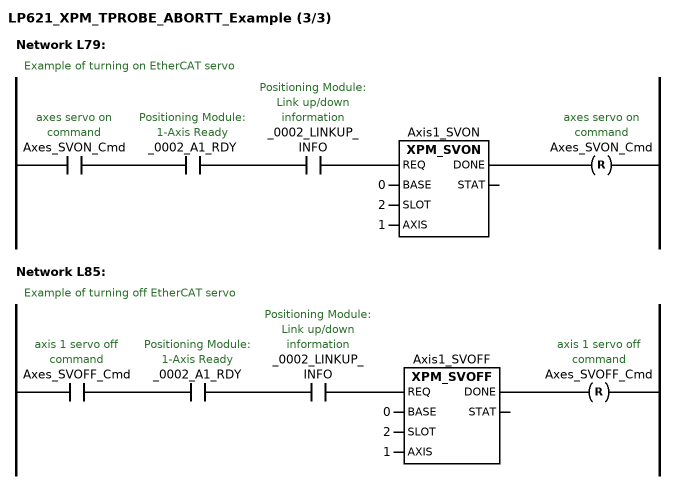
(* [picture p24: LP621_XPM_TPROBE_ABORTT_Example rungs L79-L85] *)
(* Example of turning on EtherCAT servo *)
(* Rung L79 *)
Axis1_SVON(REQ := Axes_SVON_Cmd AND _0002_A1_RDY AND _0002_LINKUP_INFO, BASE := 0, SLOT := 2, AXIS := 1);
IF Axis1_SVON.DONE THEN Axes_SVON_Cmd := FALSE; END_IF;
(* Example of turning off EtherCAT servo *)
(* Rung L85 *)
Axis1_SVOFF(REQ := Axes_SVOFF_Cmd AND _0002_A1_RDY AND _0002_LINKUP_INFO, BASE := 0, SLOT := 2, AXIS := 1);
IF Axis1_SVOFF.DONE THEN Axes_SVOFF_Cmd := FALSE; END_IF;
END_PROGRAM

PROGRAM LP622_Read_Data_Example (* task: Scan Program *)
(* example program for XPM_CRD and XPM_SRD function blocks. *)
VAR
    Axes_SVOFF_Cmd : BOOL; (* axis 1 servo off command *)
    Axes_SVON_Cmd : BOOL; (* axes servo on command *)
    Axis1_Commanded_Position : DINT; (* commanded position of axis 1 *)
    Axis1_Commanded_Speed : DINT; (* commanded speed of axis 1 *)
    Axis1_CommonError_Number : UINT; (* common error number for axis 1 *)
    Axis1_CRD : XPM_CRD; (* axis 1 drive information fb *)
    Axis1_Current_Position : DINT; (* current position of axis 1 *)
    Axis1_Current_Speed : DINT; (* current speed of axis 1 *)
    Axis1_Current_Step : UINT; (* current position table step of axis 1 *)
    Axis1_Current_Torque : INT; (* current torque of axis 1 *)
    Axis1_Error_Number : UINT; (* error number for axis 1 *)
    Axis1_MCode : UINT; (* axis1 mcode *)
    Axis1_Read_Data : BOOL; (* command to read axis data *)
    Axis1_SRD : XPM_SRD; (* axis 1 state function block *)
    Axis1_ST1 : ARRAY[0..7] OF BOOL; (* axis 1 state 1 information *)
    Axis1_ST2 : ARRAY[0..7] OF BOOL; (* axis 1 state 2 information *)
    Axis1_ST3 : ARRAY[0..7] OF BOOL; (* axis 1 state 3 information *)
    Axis1_ST4 : ARRAY[0..7] OF BOOL; (* axis 1 state 4 information *)
    Axis1_ST5 : ARRAY[0..7] OF BOOL; (* axis 1 state 5 information *)
    Axis1_ST6 : ARRAY[0..7] OF BOOL; (* axis 1 state 6 information *)
    Axis1_ST7 : ARRAY[0..7] OF BOOL; (* axis 1 state 7 information *)
    Axis1_SVOFF : XPM_SVOFF; (* function block for axis 1 servo off *)
    Axis1_SVON : XPM_SVON; (* SVON fb for axis 1 *)
    Connect_Servos : BOOL; (* command to connect to ECAT servos *)
    DCON_FB : XPM_DCON; (* EtherCAT disconnect FB *)
    Disconnect_Servos : BOOL; (* Disconnect from ECAT servos *)
    ECON_FB : XPM_ECON; (* EtherCAT connect FB *)
END_VAR
VAR_EXTERNAL
    _0002_A1_RDY : BOOL; (* AT %UX0.2.0 *) (* Positioning Module: 1-Axis Ready *)
    _0002_LINKUP_INFO : BOOL; (* AT %UX0.2.14 *) (* Positioning Module: Link up/down information *)
END_VAR

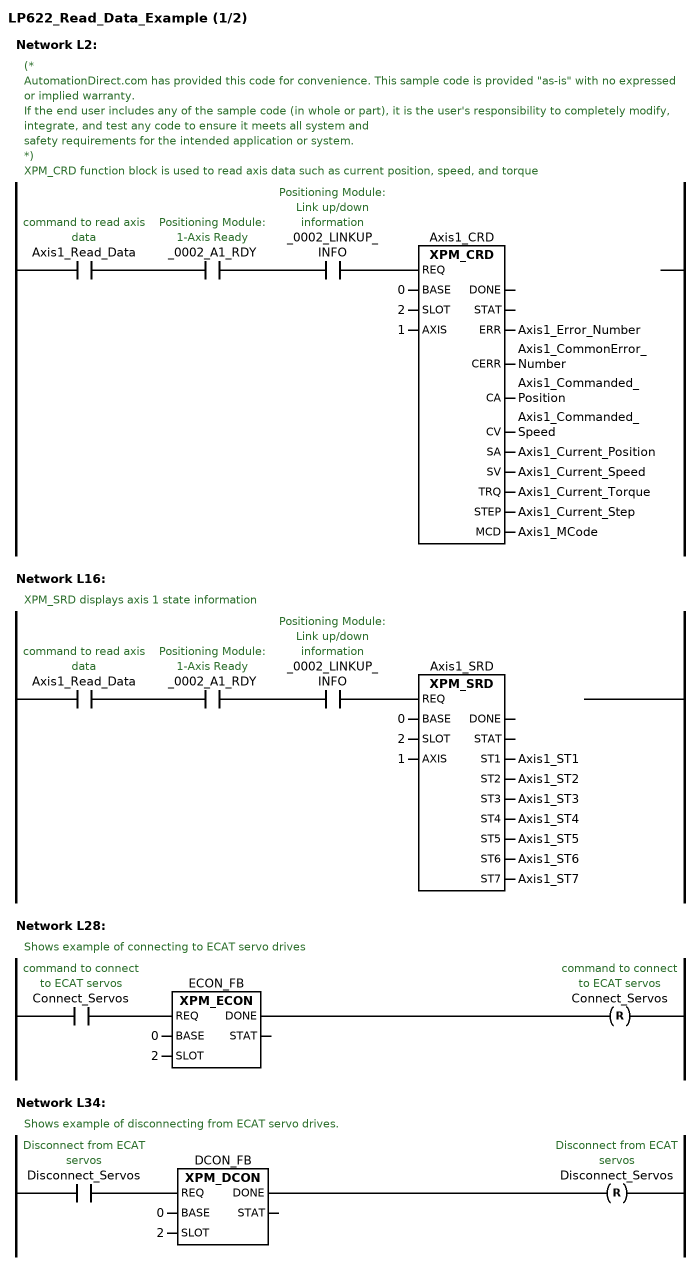
(* ( * / AutomationDirect.com has provided this code for convenience. This sample code is provided "as-is" with no expressed or implied warranty. / If the end user includes any of the sample code (in whole or part), it is the user's responsibility to completely modify, integrate, and test any code to ensure it meets all system and / safety requirements for the intended application or system. / * ) *)
(* XPM_CRD function block is used to read axis data such as current position, speed, and torque *)
(* Rung L2 *)
Axis1_CRD(REQ := Axis1_Read_Data AND _0002_A1_RDY AND _0002_LINKUP_INFO, BASE := 0, SLOT := 2, AXIS := 1, ERR => Axis1_Error_Number, CERR => Axis1_CommonError_Number, CA => Axis1_Commanded_Position, CV => Axis1_Commanded_Speed, SA => Axis1_Current_Position, SV => Axis1_Current_Speed, TRQ => Axis1_Current_Torque, STEP => Axis1_Current_Step, MCD => Axis1_MCode);
(* XPM_SRD displays axis 1 state information *)
(* Rung L16 *)
Axis1_SRD(REQ := Axis1_Read_Data AND _0002_A1_RDY AND _0002_LINKUP_INFO, BASE := 0, SLOT := 2, AXIS := 1, ST1 => Axis1_ST1, ST2 => Axis1_ST2, ST3 => Axis1_ST3, ST4 => Axis1_ST4, ST5 => Axis1_ST5, ST6 => Axis1_ST6, ST7 => Axis1_ST7);
(* Shows example of connecting to ECAT servo drives *)
(* Rung L28 *)
ECON_FB(REQ := Connect_Servos, BASE := 0, SLOT := 2);
IF ECON_FB.DONE THEN Connect_Servos := FALSE; END_IF;
(* Shows example of disconnecting from ECAT servo drives. *)
(* Rung L34 *)
DCON_FB(REQ := Disconnect_Servos, BASE := 0, SLOT := 2);
IF DCON_FB.DONE THEN Disconnect_Servos := FALSE; END_IF;

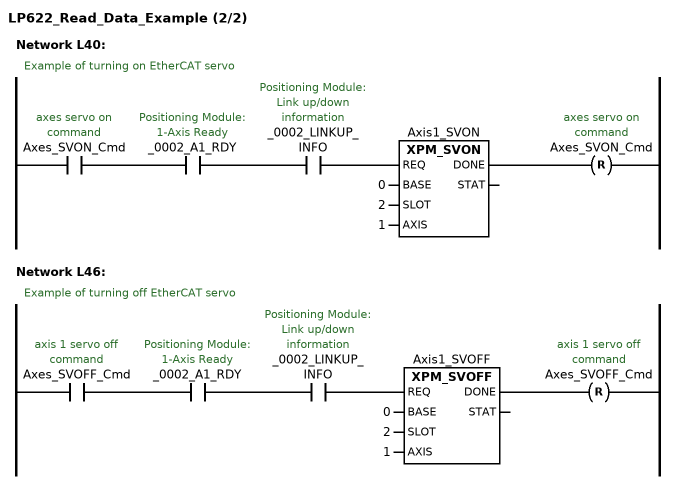
(* Example of turning on EtherCAT servo *)
(* Rung L40 *)
Axis1_SVON(REQ := Axes_SVON_Cmd AND _0002_A1_RDY AND _0002_LINKUP_INFO, BASE := 0, SLOT := 2, AXIS := 1);
IF Axis1_SVON.DONE THEN Axes_SVON_Cmd := FALSE; END_IF;
(* Example of turning off EtherCAT servo *)
(* Rung L46 *)
Axis1_SVOFF(REQ := Axes_SVOFF_Cmd AND _0002_A1_RDY AND _0002_LINKUP_INFO, BASE := 0, SLOT := 2, AXIS := 1);
IF Axis1_SVOFF.DONE THEN Axes_SVOFF_Cmd := FALSE; END_IF;
END_PROGRAM

PROGRAM LP624_XPM_JOG_Example (* task: Scan Program *)
(* example program for XPM_JOG and XPM_RTP function block. *)
VAR
    Axes_SVOFF_Cmd : BOOL; (* axis 1 servo off command *)
    Axes_SVON_Cmd : BOOL; (* axes servo on command *)
    Axis1_Home : XPM_FLT; (* direct home of axis 1 *)
    Axis1_Jog_FWD : XPM_JOG; (* fb to jog axis 1 fwd *)
    Axis1_Jog_FWD_CMD : BOOL; (* command to jog axis 1 forward *)
    Axis1_Jog_REV : XPM_JOG; (* axis 1 jog reverse fb *)
    Axis1_Jog_REV_CMD : BOOL; (* command to jog axis 1 in reverse *)
    Axis1_RTP : XPM_RTP; (* axis 1 return to position fb *)
    Axis1_RTP_CMD : BOOL; (* return axis 1 to position before manual move *)
    Axis1_SVOFF : XPM_SVOFF; (* function block for axis 1 servo off *)
    Axis1_SVON : XPM_SVON; (* SVON fb for axis 1 *)
    Axis2_Jog_FWD : XPM_JOG; (* fb to jog axis 1 fwd *)
    Connect_Servos : BOOL; (* command to connect to ECAT servos *)
    DCON_FB : XPM_DCON; (* EtherCAT disconnect FB *)
    Disconnect_Servos : BOOL; (* Disconnect from ECAT servos *)
    ECON_FB : XPM_ECON; (* EtherCAT connect FB *)
    Home_Axes : BOOL; (* home the axes *)
END_VAR
VAR_EXTERNAL
    _0002_A1_RDY : BOOL; (* AT %UX0.2.0 *) (* Positioning Module: 1-Axis Ready *)
    _0002_A4_RDY : BOOL; (* AT %UX0.2.3 *) (* Positioning Module: 4-Axis Ready *)
    _0002_LINKUP_INFO : BOOL; (* AT %UX0.2.14 *) (* Positioning Module: Link up/down information *)
END_VAR

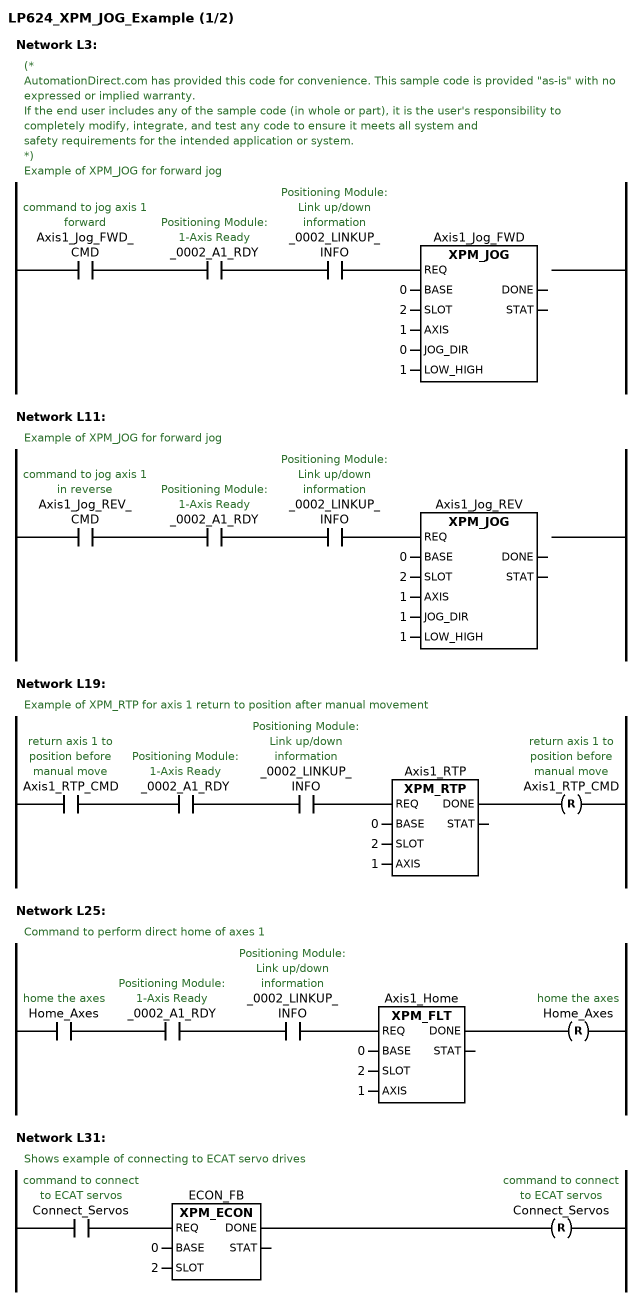
(* ( * / AutomationDirect.com has provided this code for convenience. This sample code is provided "as-is" with no expressed or implied warranty. / If the end user includes any of the sample code (in whole or part), it is the user's responsibility to completely modify, integrate, and test any code to ensure it meets all system and / safety requirements for the intended application or system. / * ) *)
(* Example of XPM_JOG for forward jog *)
(* Rung L3 *)
Axis1_Jog_FWD(REQ := Axis1_Jog_FWD_CMD AND _0002_A1_RDY AND _0002_LINKUP_INFO, BASE := 0, SLOT := 2, AXIS := 1, JOG_DIR := 0, LOW_HIGH := 1);
(* Example of XPM_JOG for forward jog *)
(* Rung L11 *)
Axis1_Jog_REV(REQ := Axis1_Jog_REV_CMD AND _0002_A1_RDY AND _0002_LINKUP_INFO, BASE := 0, SLOT := 2, AXIS := 1, JOG_DIR := 1, LOW_HIGH := 1);
(* Example of XPM_RTP for axis 1 return to position after manual movement *)
(* Rung L19 *)
Axis1_RTP(REQ := Axis1_RTP_CMD AND _0002_A1_RDY AND _0002_LINKUP_INFO, BASE := 0, SLOT := 2, AXIS := 1);
IF Axis1_RTP.DONE THEN Axis1_RTP_CMD := FALSE; END_IF;
(* Command to perform direct home of axes 1 *)
(* Rung L25 *)
Axis1_Home(REQ := Home_Axes AND _0002_A1_RDY AND _0002_LINKUP_INFO, BASE := 0, SLOT := 2, AXIS := 1);
IF Axis1_Home.DONE THEN Home_Axes := FALSE; END_IF;
(* Shows example of connecting to ECAT servo drives *)
(* Rung L31 *)
ECON_FB(REQ := Connect_Servos, BASE := 0, SLOT := 2);
IF ECON_FB.DONE THEN Connect_Servos := FALSE; END_IF;

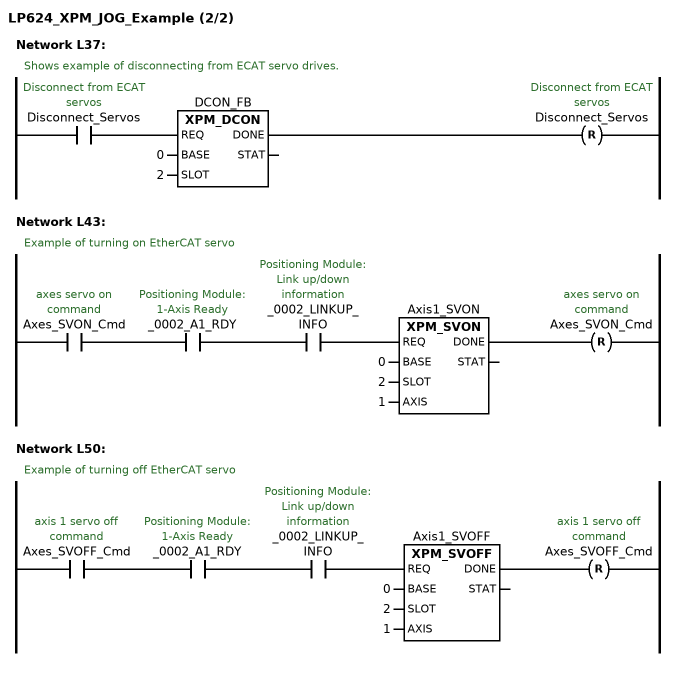
(* Shows example of disconnecting from ECAT servo drives. *)
(* Rung L37 *)
DCON_FB(REQ := Disconnect_Servos, BASE := 0, SLOT := 2);
IF DCON_FB.DONE THEN Disconnect_Servos := FALSE; END_IF;
(* Example of turning on EtherCAT servo *)
(* Rung L43 *)
Axis1_SVON(REQ := Axes_SVON_Cmd AND _0002_A1_RDY AND _0002_LINKUP_INFO, BASE := 0, SLOT := 2, AXIS := 1);
IF Axis1_SVON.DONE THEN Axes_SVON_Cmd := FALSE; END_IF;
(* Example of turning off EtherCAT servo *)
(* Rung L50 *)
Axis1_SVOFF(REQ := Axes_SVOFF_Cmd AND _0002_A1_RDY AND _0002_LINKUP_INFO, BASE := 0, SLOT := 2, AXIS := 1);
IF Axis1_SVOFF.DONE THEN Axes_SVOFF_Cmd := FALSE; END_IF;
END_PROGRAM

PROGRAM LP625_XPM_INC_Example (* task: Scan Program *)
(* example program for XPM_INC and XPM_RTP function block. *)
VAR
    Axes_SVOFF_Cmd : BOOL; (* axis 1 servo off command *)
    Axes_SVON_Cmd : BOOL; (* axes servo on command *)
    Axis1_Home : XPM_FLT; (* direct home of axis 1 *)
    Axis1_Inch_CMD : BOOL; (* command to jog axis 1 forward *)
    Axis1_Inch_FB : XPM_INC; (* inching fb for axis 1 *)
    Axis1_Inch_Value : DINT; (* inching value for axis 1 *)
    Axis1_RTP : XPM_RTP; (* axis 1 return to position fb *)
    Axis1_RTP_CMD : BOOL; (* return axis 1 to position before manual move *)
    Axis1_SVOFF : XPM_SVOFF; (* function block for axis 1 servo off *)
    Axis1_SVON : XPM_SVON; (* SVON fb for axis 1 *)
    Connect_Servos : BOOL; (* command to connect to ECAT servos *)
    DCON_FB : XPM_DCON; (* EtherCAT disconnect FB *)
    Disconnect_Servos : BOOL; (* Disconnect from ECAT servos *)
    ECON_FB : XPM_ECON; (* EtherCAT connect FB *)
    Home_Axes : BOOL; (* home the axes *)
END_VAR
VAR_EXTERNAL
    _0002_A1_RDY : BOOL; (* AT %UX0.2.0 *) (* Positioning Module: 1-Axis Ready *)
    _0002_LINKUP_INFO : BOOL; (* AT %UX0.2.14 *) (* Positioning Module: Link up/down information *)
END_VAR

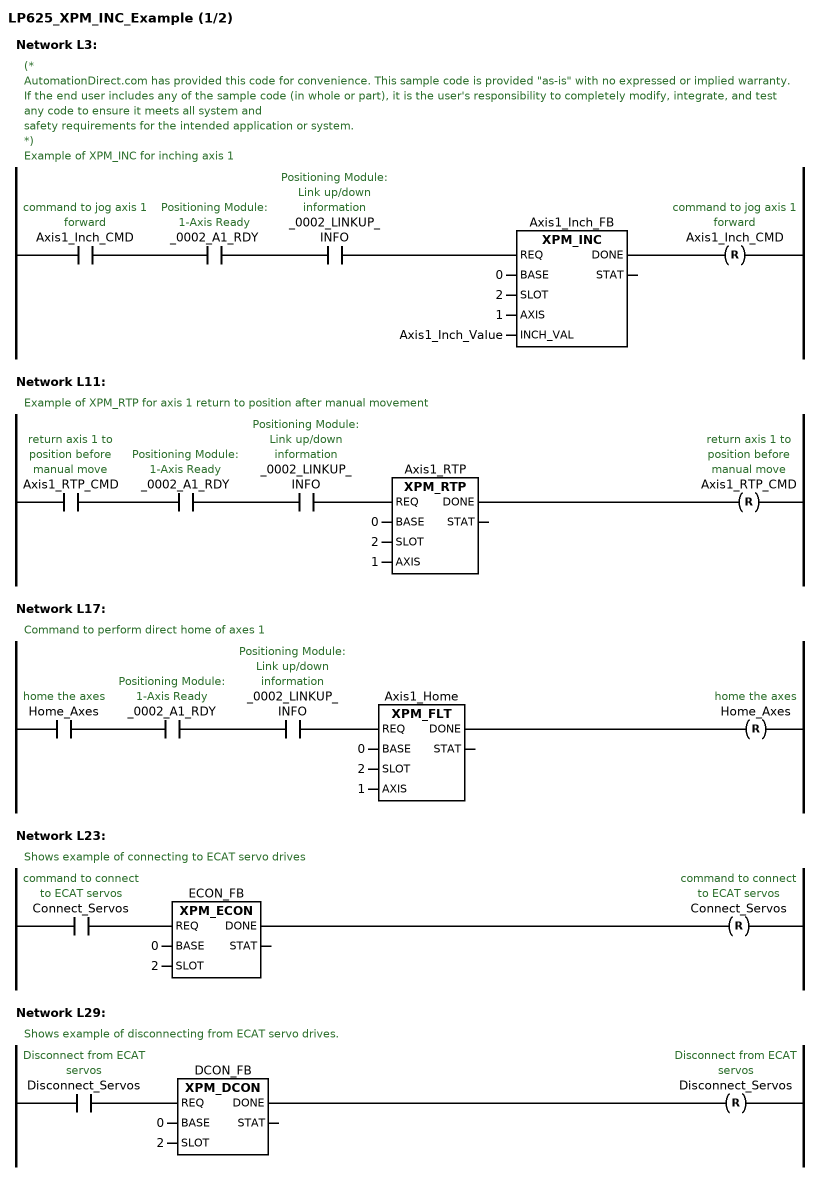
(* ( * / AutomationDirect.com has provided this code for convenience. This sample code is provided "as-is" with no expressed or implied warranty. / If the end user includes any of the sample code (in whole or part), it is the user's responsibility to completely modify, integrate, and test any code to ensure it meets all system and / safety requirements for the intended application or system. / * ) *)
(* Example of XPM_INC for inching axis 1 *)
(* Rung L3 *)
Axis1_Inch_FB(REQ := Axis1_Inch_CMD AND _0002_A1_RDY AND _0002_LINKUP_INFO, BASE := 0, SLOT := 2, AXIS := 1, INCH_VAL := Axis1_Inch_Value);
IF Axis1_Inch_FB.DONE THEN Axis1_Inch_CMD := FALSE; END_IF;
(* Example of XPM_RTP for axis 1 return to position after manual movement *)
(* Rung L11 *)
Axis1_RTP(REQ := Axis1_RTP_CMD AND _0002_A1_RDY AND _0002_LINKUP_INFO, BASE := 0, SLOT := 2, AXIS := 1);
IF Axis1_RTP.DONE THEN Axis1_RTP_CMD := FALSE; END_IF;
(* Command to perform direct home of axes 1 *)
(* Rung L17 *)
Axis1_Home(REQ := Home_Axes AND _0002_A1_RDY AND _0002_LINKUP_INFO, BASE := 0, SLOT := 2, AXIS := 1);
IF Axis1_Home.DONE THEN Home_Axes := FALSE; END_IF;
(* Shows example of connecting to ECAT servo drives *)
(* Rung L23 *)
ECON_FB(REQ := Connect_Servos, BASE := 0, SLOT := 2);
IF ECON_FB.DONE THEN Connect_Servos := FALSE; END_IF;
(* Shows example of disconnecting from ECAT servo drives. *)
(* Rung L29 *)
DCON_FB(REQ := Disconnect_Servos, BASE := 0, SLOT := 2);
IF DCON_FB.DONE THEN Disconnect_Servos := FALSE; END_IF;

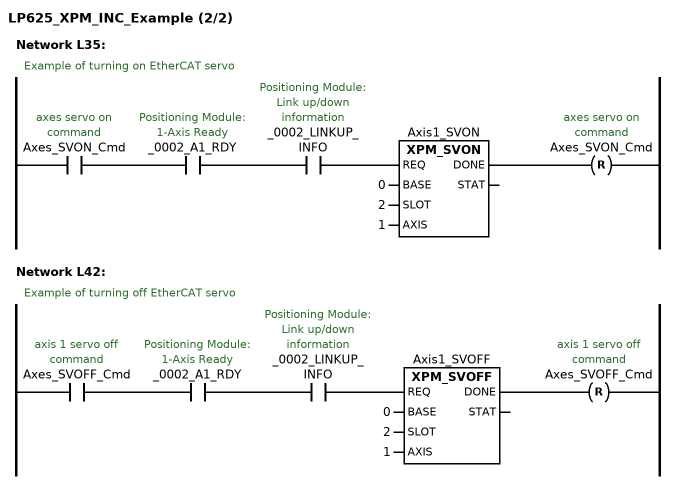
(* Example of turning on EtherCAT servo *)
(* Rung L35 *)
Axis1_SVON(REQ := Axes_SVON_Cmd AND _0002_A1_RDY AND _0002_LINKUP_INFO, BASE := 0, SLOT := 2, AXIS := 1);
IF Axis1_SVON.DONE THEN Axes_SVON_Cmd := FALSE; END_IF;
(* Example of turning off EtherCAT servo *)
(* Rung L42 *)
Axis1_SVOFF(REQ := Axes_SVOFF_Cmd AND _0002_A1_RDY AND _0002_LINKUP_INFO, BASE := 0, SLOT := 2, AXIS := 1);
IF Axis1_SVOFF.DONE THEN Axes_SVOFF_Cmd := FALSE; END_IF;
END_PROGRAM

PROGRAM LP626_Homing_Example (* task: Scan Program *)
(* example program for XPM_ORG and XPM_FLT  function block. *)
VAR
    Axes_SVOFF_Cmd : BOOL; (* axis 1 servo off command *)
    Axes_SVON_Cmd : BOOL; (* axes servo on command *)
    Axis1_FLT_CMD : BOOL; (* home axis 1 with XPM_FLT *)
    Axis1_ORG_CMD : BOOL; (* home axis 1 with XPM_ORG *)
    Axis1_SVOFF : XPM_SVOFF; (* function block for axis 1 servo off *)
    Axis1_SVON : XPM_SVON; (* SVON fb for axis 1 *)
    Axis1_XPM_FLT : XPM_FLT; (* direct home of axis 1 *)
    Axis1_XPM_ORG : XPM_ORG; (* axis 1 xpm_org fb *)
    Connect_Servos : BOOL; (* command to connect to ECAT servos *)
    DCON_FB : XPM_DCON; (* EtherCAT disconnect FB *)
    Disconnect_Servos : BOOL; (* Disconnect from ECAT servos *)
    ECON_FB : XPM_ECON; (* EtherCAT connect FB *)
END_VAR
VAR_EXTERNAL
    _0002_A1_RDY : BOOL; (* AT %UX0.2.0 *) (* Positioning Module: 1-Axis Ready *)
    _0002_LINKUP_INFO : BOOL; (* AT %UX0.2.14 *) (* Positioning Module: Link up/down information *)
END_VAR

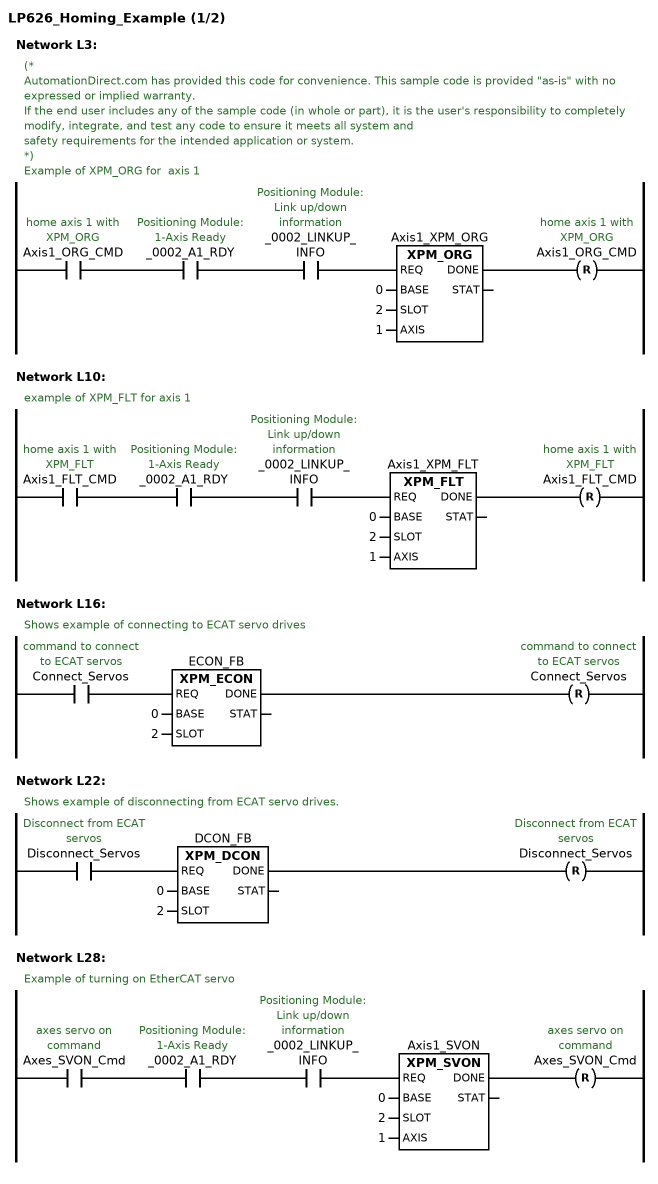
(* ( * / AutomationDirect.com has provided this code for convenience. This sample code is provided "as-is" with no expressed or implied warranty. / If the end user includes any of the sample code (in whole or part), it is the user's responsibility to completely modify, integrate, and test any code to ensure it meets all system and / safety requirements for the intended application or system. / * ) *)
(* Example of XPM_ORG for  axis 1 *)
(* Rung L3 *)
Axis1_XPM_ORG(REQ := Axis1_ORG_CMD AND _0002_A1_RDY AND _0002_LINKUP_INFO, BASE := 0, SLOT := 2, AXIS := 1);
IF Axis1_XPM_ORG.DONE THEN Axis1_ORG_CMD := FALSE; END_IF;
(* example of XPM_FLT for axis 1 *)
(* Rung L10 *)
Axis1_XPM_FLT(REQ := Axis1_FLT_CMD AND _0002_A1_RDY AND _0002_LINKUP_INFO, BASE := 0, SLOT := 2, AXIS := 1);
IF Axis1_XPM_FLT.DONE THEN Axis1_FLT_CMD := FALSE; END_IF;
(* Shows example of connecting to ECAT servo drives *)
(* Rung L16 *)
ECON_FB(REQ := Connect_Servos, BASE := 0, SLOT := 2);
IF ECON_FB.DONE THEN Connect_Servos := FALSE; END_IF;
(* Shows example of disconnecting from ECAT servo drives. *)
(* Rung L22 *)
DCON_FB(REQ := Disconnect_Servos, BASE := 0, SLOT := 2);
IF DCON_FB.DONE THEN Disconnect_Servos := FALSE; END_IF;
(* Example of turning on EtherCAT servo *)
(* Rung L28 *)
Axis1_SVON(REQ := Axes_SVON_Cmd AND _0002_A1_RDY AND _0002_LINKUP_INFO, BASE := 0, SLOT := 2, AXIS := 1);
IF Axis1_SVON.DONE THEN Axes_SVON_Cmd := FALSE; END_IF;

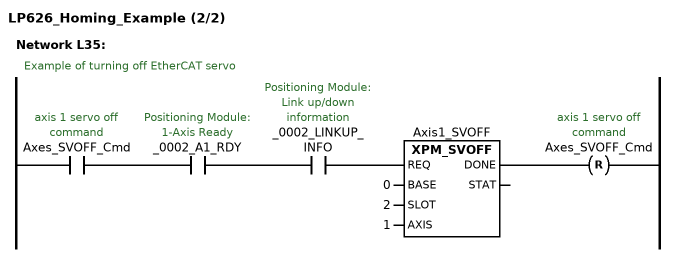
(* Example of turning off EtherCAT servo *)
(* Rung L35 *)
Axis1_SVOFF(REQ := Axes_SVOFF_Cmd AND _0002_A1_RDY AND _0002_LINKUP_INFO, BASE := 0, SLOT := 2, AXIS := 1);
IF Axis1_SVOFF.DONE THEN Axes_SVOFF_Cmd := FALSE; END_IF;
END_PROGRAM

PROGRAM LP627_XPM_DST_Example (* task: Scan Program *)
(* example program for XPM_DST  function block. *)
VAR
    Axes_SVOFF_Cmd : BOOL; (* axis 1 servo off command *)
    Axes_SVON_Cmd : BOOL; (* axes servo on command *)
    Axis1_ABSINC : BOOL;
    Axis1_ADDR : DINT; (* axis 1 addr input value *)
    Axis1_CTRL : USINT;
    Axis1_DST_CMD : BOOL; (* command to jog axis 1 forward *)
    Axis1_DST_FB : XPM_DST; (* xpm_dst for axis 1 *)
    Axis1_DWELL : UINT;
    Axis1_Home : XPM_FLT; (* direct home of axis 1 *)
    Axis1_SPEED : UDINT;
    Axis1_SVOFF : XPM_SVOFF; (* function block for axis 1 servo off *)
    Axis1_SVON : XPM_SVON; (* SVON fb for axis 1 *)
    Connect_Servos : BOOL; (* command to connect to ECAT servos *)
    DCON_FB : XPM_DCON; (* EtherCAT disconnect FB *)
    Disconnect_Servos : BOOL; (* Disconnect from ECAT servos *)
    ECON_FB : XPM_ECON; (* EtherCAT connect FB *)
    Home_Axes : BOOL; (* home the axes *)
END_VAR
VAR_EXTERNAL
    _0002_A1_RDY : BOOL; (* AT %UX0.2.0 *) (* Positioning Module: 1-Axis Ready *)
    _0002_LINKUP_INFO : BOOL; (* AT %UX0.2.14 *) (* Positioning Module: Link up/down information *)
END_VAR

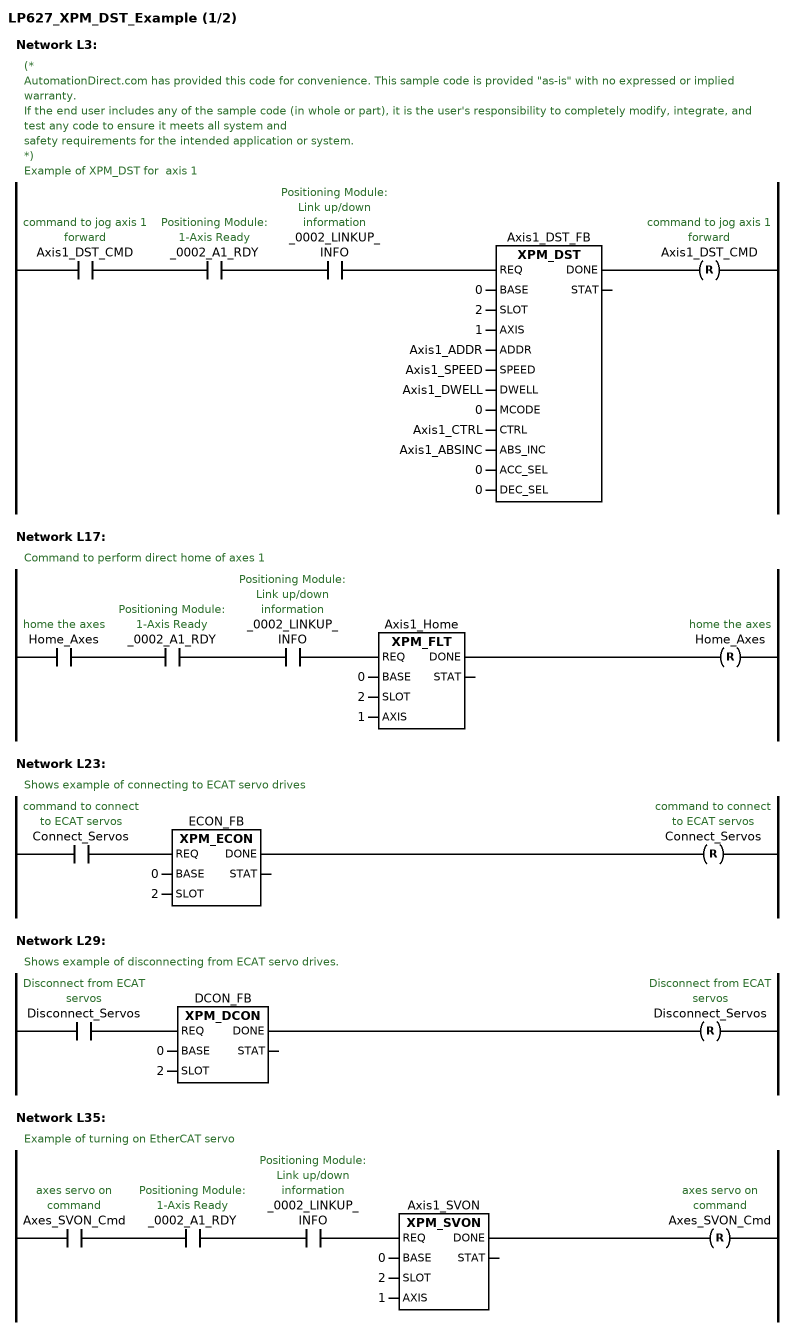
(* ( * / AutomationDirect.com has provided this code for convenience. This sample code is provided "as-is" with no expressed or implied warranty. / If the end user includes any of the sample code (in whole or part), it is the user's responsibility to completely modify, integrate, and test any code to ensure it meets all system and / safety requirements for the intended application or system. / * ) *)
(* Example of XPM_DST for  axis 1 *)
(* Rung L3 *)
Axis1_DST_FB(REQ := Axis1_DST_CMD AND _0002_A1_RDY AND _0002_LINKUP_INFO, BASE := 0, SLOT := 2, AXIS := 1, ADDR := Axis1_ADDR, SPEED := Axis1_SPEED, DWELL := Axis1_DWELL, MCODE := 0, CTRL := Axis1_CTRL, ABS_INC := Axis1_ABSINC, ACC_SEL := 0, DEC_SEL := 0);
IF Axis1_DST_FB.DONE THEN Axis1_DST_CMD := FALSE; END_IF;
(* Command to perform direct home of axes 1 *)
(* Rung L17 *)
Axis1_Home(REQ := Home_Axes AND _0002_A1_RDY AND _0002_LINKUP_INFO, BASE := 0, SLOT := 2, AXIS := 1);
IF Axis1_Home.DONE THEN Home_Axes := FALSE; END_IF;
(* Shows example of connecting to ECAT servo drives *)
(* Rung L23 *)
ECON_FB(REQ := Connect_Servos, BASE := 0, SLOT := 2);
IF ECON_FB.DONE THEN Connect_Servos := FALSE; END_IF;
(* Shows example of disconnecting from ECAT servo drives. *)
(* Rung L29 *)
DCON_FB(REQ := Disconnect_Servos, BASE := 0, SLOT := 2);
IF DCON_FB.DONE THEN Disconnect_Servos := FALSE; END_IF;
(* Example of turning on EtherCAT servo *)
(* Rung L35 *)
Axis1_SVON(REQ := Axes_SVON_Cmd AND _0002_A1_RDY AND _0002_LINKUP_INFO, BASE := 0, SLOT := 2, AXIS := 1);
IF Axis1_SVON.DONE THEN Axes_SVON_Cmd := FALSE; END_IF;

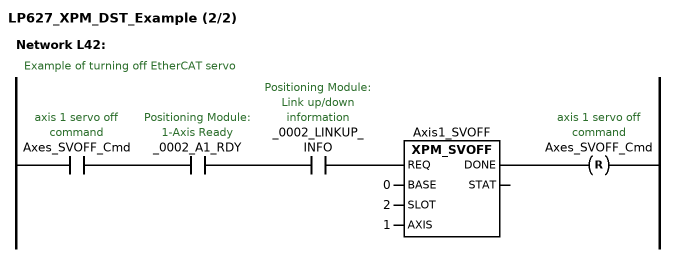
(* Example of turning off EtherCAT servo *)
(* Rung L42 *)
Axis1_SVOFF(REQ := Axes_SVOFF_Cmd AND _0002_A1_RDY AND _0002_LINKUP_INFO, BASE := 0, SLOT := 2, AXIS := 1);
IF Axis1_SVOFF.DONE THEN Axes_SVOFF_Cmd := FALSE; END_IF;
END_PROGRAM

PROGRAM LP628_XPM_IST_Example (* task: Scan Program *)
(* example program for XPM_IST  function block. *)
VAR
    Axes_SVOFF_Cmd : BOOL; (* axis 1 servo off command *)
    Axes_SVON_Cmd : BOOL; (* axes servo on command *)
    Axis1_CMD_Step : UINT; (* step to run in XPM_IST *)
    Axis1_Home : XPM_FLT; (* direct home of axis 1 *)
    Axis1_IST_CMD : BOOL; (* command to jog axis 1 forward *)
    Axis1_IST_FB : XPM_IST; (* xpm_ist for axis 1 *)
    Axis1_SVOFF : XPM_SVOFF; (* function block for axis 1 servo off *)
    Axis1_SVON : XPM_SVON; (* SVON fb for axis 1 *)
    Connect_Servos : BOOL; (* command to connect to ECAT servos *)
    DCON_FB : XPM_DCON; (* EtherCAT disconnect FB *)
    Disconnect_Servos : BOOL; (* Disconnect from ECAT servos *)
    ECON_FB : XPM_ECON; (* EtherCAT connect FB *)
    Home_Axes : BOOL; (* home the axes *)
END_VAR
VAR_EXTERNAL
    _0002_A1_RDY : BOOL; (* AT %UX0.2.0 *) (* Positioning Module: 1-Axis Ready *)
    _0002_LINKUP_INFO : BOOL; (* AT %UX0.2.14 *) (* Positioning Module: Link up/down information *)
END_VAR

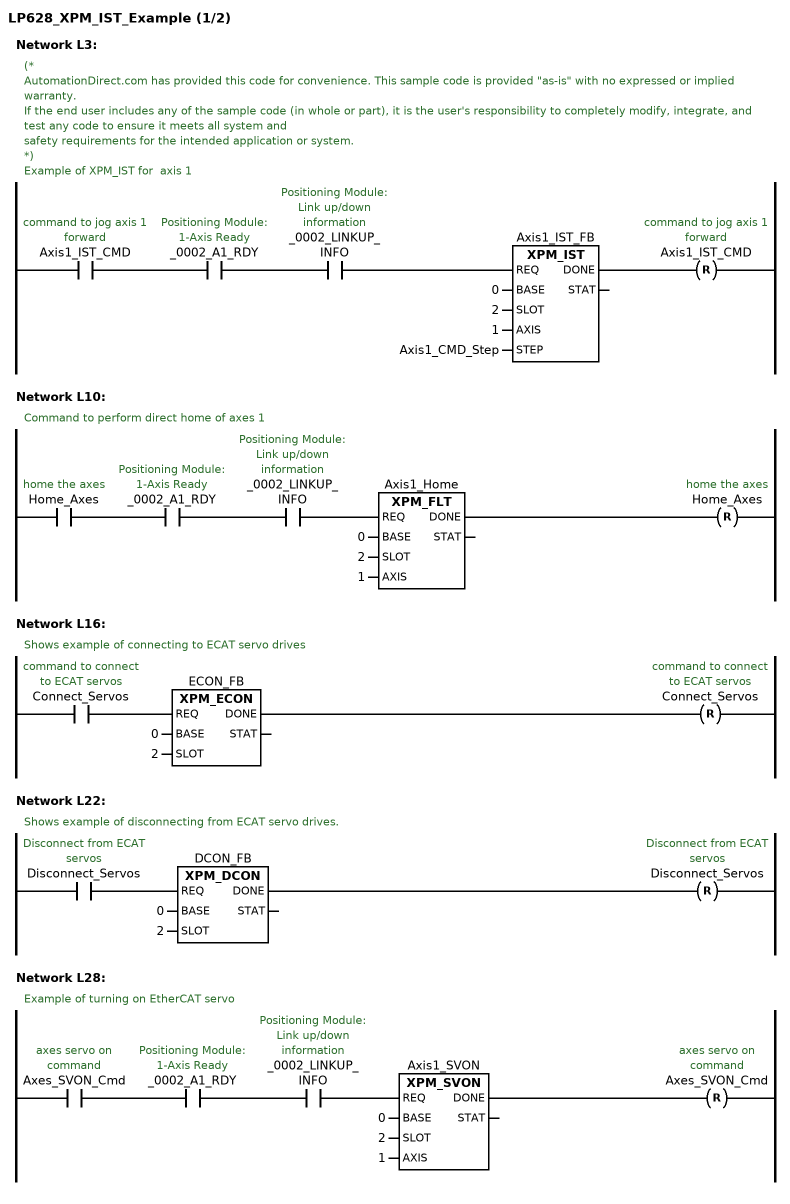
(* ( * / AutomationDirect.com has provided this code for convenience. This sample code is provided "as-is" with no expressed or implied warranty. / If the end user includes any of the sample code (in whole or part), it is the user's responsibility to completely modify, integrate, and test any code to ensure it meets all system and / safety requirements for the intended application or system. / * ) *)
(* Example of XPM_IST for  axis 1 *)
(* Rung L3 *)
Axis1_IST_FB(REQ := Axis1_IST_CMD AND _0002_A1_RDY AND _0002_LINKUP_INFO, BASE := 0, SLOT := 2, AXIS := 1, STEP := Axis1_CMD_Step);
IF Axis1_IST_FB.DONE THEN Axis1_IST_CMD := FALSE; END_IF;
(* Command to perform direct home of axes 1 *)
(* Rung L10 *)
Axis1_Home(REQ := Home_Axes AND _0002_A1_RDY AND _0002_LINKUP_INFO, BASE := 0, SLOT := 2, AXIS := 1);
IF Axis1_Home.DONE THEN Home_Axes := FALSE; END_IF;
(* Shows example of connecting to ECAT servo drives *)
(* Rung L16 *)
ECON_FB(REQ := Connect_Servos, BASE := 0, SLOT := 2);
IF ECON_FB.DONE THEN Connect_Servos := FALSE; END_IF;
(* Shows example of disconnecting from ECAT servo drives. *)
(* Rung L22 *)
DCON_FB(REQ := Disconnect_Servos, BASE := 0, SLOT := 2);
IF DCON_FB.DONE THEN Disconnect_Servos := FALSE; END_IF;
(* Example of turning on EtherCAT servo *)
(* Rung L28 *)
Axis1_SVON(REQ := Axes_SVON_Cmd AND _0002_A1_RDY AND _0002_LINKUP_INFO, BASE := 0, SLOT := 2, AXIS := 1);
IF Axis1_SVON.DONE THEN Axes_SVON_Cmd := FALSE; END_IF;

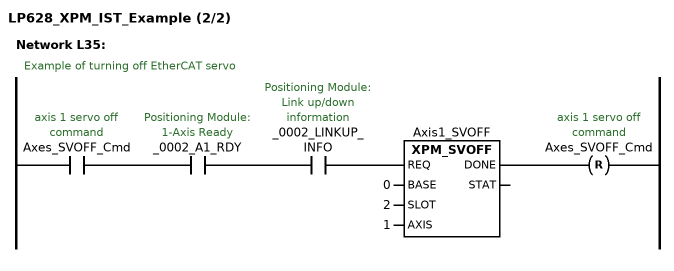
(* Example of turning off EtherCAT servo *)
(* Rung L35 *)
Axis1_SVOFF(REQ := Axes_SVOFF_Cmd AND _0002_A1_RDY AND _0002_LINKUP_INFO, BASE := 0, SLOT := 2, AXIS := 1);
IF Axis1_SVOFF.DONE THEN Axes_SVOFF_Cmd := FALSE; END_IF;
END_PROGRAM

PROGRAM LP629_XPM_RST_Example (* task: Scan Program *)
(* example program for XPM_RST  function block. *)
VAR
    Axes_SVOFF_Cmd : BOOL; (* axis 1 servo off command *)
    Axes_SVON_Cmd : BOOL; (* axes servo on command *)
    Axis1_RST : XPM_RST; (* xpm_rst function block *)
    Axis1_RST_CMD : BOOL; (* command to jog axis 1 forward *)
    Axis1_SVOFF : XPM_SVOFF; (* function block for axis 1 servo off *)
    Axis1_SVON : XPM_SVON; (* SVON fb for axis 1 *)
    Connect_Servos : BOOL; (* command to connect to ECAT servos *)
    DCON_FB : XPM_DCON; (* EtherCAT disconnect FB *)
    Disconnect_Servos : BOOL; (* Disconnect from ECAT servos *)
    ECON_FB : XPM_ECON; (* EtherCAT connect FB *)
    Home_Axes : BOOL; (* home the axes *)
END_VAR
VAR_EXTERNAL
    _0002_A1_RDY : BOOL; (* AT %UX0.2.0 *) (* Positioning Module: 1-Axis Ready *)
    _0002_LINKUP_INFO : BOOL; (* AT %UX0.2.14 *) (* Positioning Module: Link up/down information *)
END_VAR

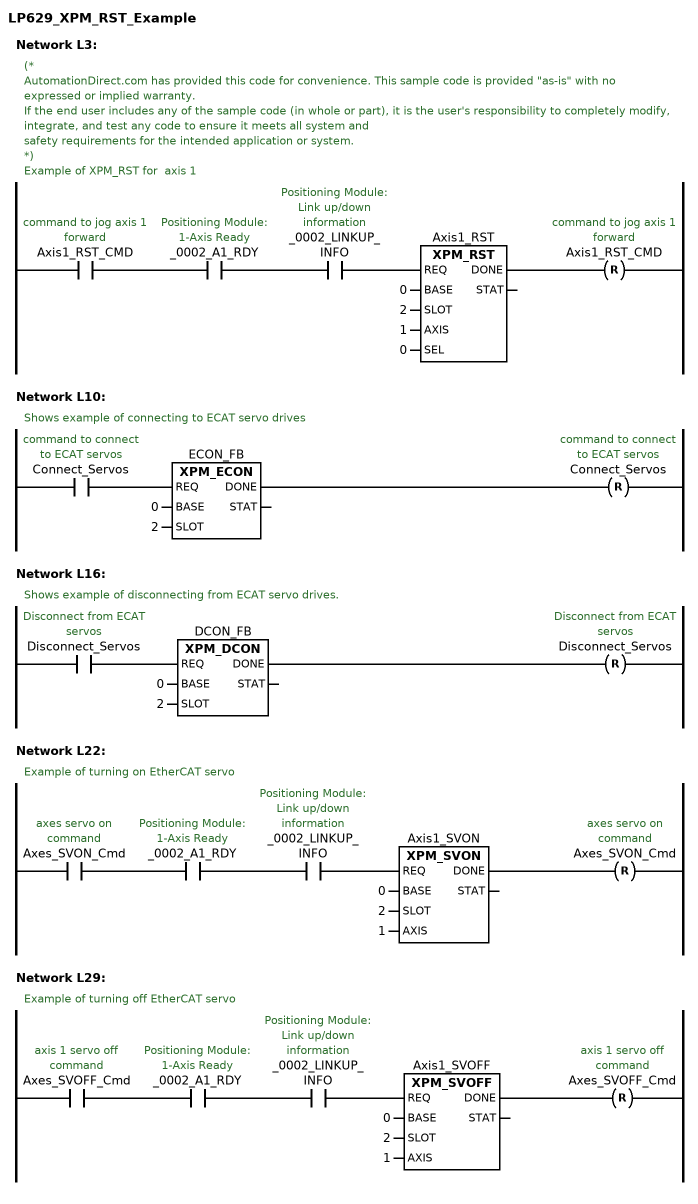
(* ( * / AutomationDirect.com has provided this code for convenience. This sample code is provided "as-is" with no expressed or implied warranty. / If the end user includes any of the sample code (in whole or part), it is the user's responsibility to completely modify, integrate, and test any code to ensure it meets all system and / safety requirements for the intended application or system. / * ) *)
(* Example of XPM_RST for  axis 1 *)
(* Rung L3 *)
Axis1_RST(REQ := Axis1_RST_CMD AND _0002_A1_RDY AND _0002_LINKUP_INFO, BASE := 0, SLOT := 2, AXIS := 1, SEL := 0);
IF Axis1_RST.DONE THEN Axis1_RST_CMD := FALSE; END_IF;
(* Shows example of connecting to ECAT servo drives *)
(* Rung L10 *)
ECON_FB(REQ := Connect_Servos, BASE := 0, SLOT := 2);
IF ECON_FB.DONE THEN Connect_Servos := FALSE; END_IF;
(* Shows example of disconnecting from ECAT servo drives. *)
(* Rung L16 *)
DCON_FB(REQ := Disconnect_Servos, BASE := 0, SLOT := 2);
IF DCON_FB.DONE THEN Disconnect_Servos := FALSE; END_IF;
(* Example of turning on EtherCAT servo *)
(* Rung L22 *)
Axis1_SVON(REQ := Axes_SVON_Cmd AND _0002_A1_RDY AND _0002_LINKUP_INFO, BASE := 0, SLOT := 2, AXIS := 1);
IF Axis1_SVON.DONE THEN Axes_SVON_Cmd := FALSE; END_IF;
(* Example of turning off EtherCAT servo *)
(* Rung L29 *)
Axis1_SVOFF(REQ := Axes_SVOFF_Cmd AND _0002_A1_RDY AND _0002_LINKUP_INFO, BASE := 0, SLOT := 2, AXIS := 1);
IF Axis1_SVOFF.DONE THEN Axes_SVOFF_Cmd := FALSE; END_IF;
END_PROGRAM

PROGRAM LP630_XPM_STP_EMG_Example (* task: Scan Program *)
(* example program for XPM_STP and XPM_EMG  function block. *)
VAR
    Axes_SVOFF_Cmd : BOOL; (* axis 1 servo off command *)
    Axes_SVON_Cmd : BOOL; (* axes servo on command *)
    Axis1_EMG : XPM_EMG; (* xpm_emg fb *)
    Axis1_EMG_CMD : BOOL; (* axis 1 emergency stop command *)
    Axis1_RST : XPM_RST; (* xpm_rst function block *)
    Axis1_STP : XPM_STP; (* xpm_stp function block *)
    Axis1_STP_CMD : BOOL; (* command to jog axis 1 forward *)
    Axis1_SVOFF : XPM_SVOFF; (* function block for axis 1 servo off *)
    Axis1_SVON : XPM_SVON; (* SVON fb for axis 1 *)
    Connect_Servos : BOOL; (* command to connect to ECAT servos *)
    DCON_FB : XPM_DCON; (* EtherCAT disconnect FB *)
    Disconnect_Servos : BOOL; (* Disconnect from ECAT servos *)
    ECON_FB : XPM_ECON; (* EtherCAT connect FB *)
    Home_Axes : BOOL; (* home the axes *)
END_VAR
VAR_EXTERNAL
    _0002_A1_RDY : BOOL; (* AT %UX0.2.0 *) (* Positioning Module: 1-Axis Ready *)
    _0002_LINKUP_INFO : BOOL; (* AT %UX0.2.14 *) (* Positioning Module: Link up/down information *)
END_VAR

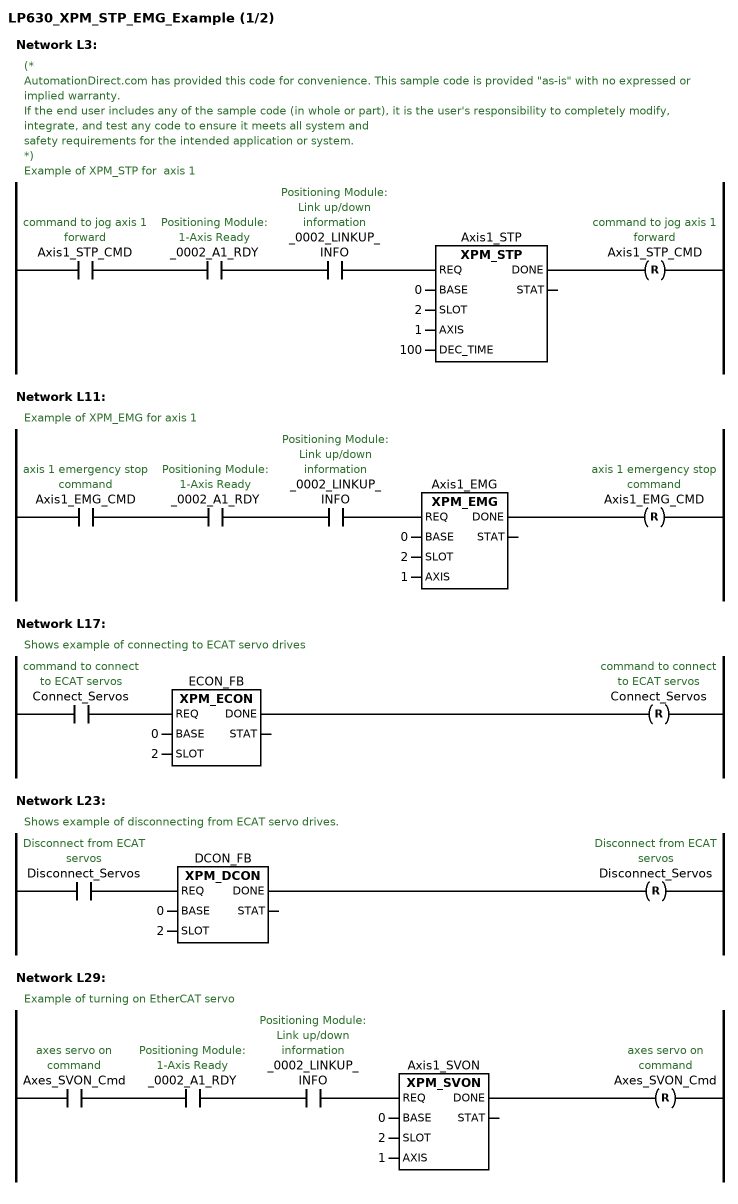
(* ( * / AutomationDirect.com has provided this code for convenience. This sample code is provided "as-is" with no expressed or implied warranty. / If the end user includes any of the sample code (in whole or part), it is the user's responsibility to completely modify, integrate, and test any code to ensure it meets all system and / safety requirements for the intended application or system. / * ) *)
(* Example of XPM_STP for  axis 1 *)
(* Rung L3 *)
Axis1_STP(REQ := Axis1_STP_CMD AND _0002_A1_RDY AND _0002_LINKUP_INFO, BASE := 0, SLOT := 2, AXIS := 1, DEC_TIME := 100);
IF Axis1_STP.DONE THEN Axis1_STP_CMD := FALSE; END_IF;
(* Example of XPM_EMG for axis 1 *)
(* Rung L11 *)
Axis1_EMG(REQ := Axis1_EMG_CMD AND _0002_A1_RDY AND _0002_LINKUP_INFO, BASE := 0, SLOT := 2, AXIS := 1);
IF Axis1_EMG.DONE THEN Axis1_EMG_CMD := FALSE; END_IF;
(* Shows example of connecting to ECAT servo drives *)
(* Rung L17 *)
ECON_FB(REQ := Connect_Servos, BASE := 0, SLOT := 2);
IF ECON_FB.DONE THEN Connect_Servos := FALSE; END_IF;
(* Shows example of disconnecting from ECAT servo drives. *)
(* Rung L23 *)
DCON_FB(REQ := Disconnect_Servos, BASE := 0, SLOT := 2);
IF DCON_FB.DONE THEN Disconnect_Servos := FALSE; END_IF;
(* Example of turning on EtherCAT servo *)
(* Rung L29 *)
Axis1_SVON(REQ := Axes_SVON_Cmd AND _0002_A1_RDY AND _0002_LINKUP_INFO, BASE := 0, SLOT := 2, AXIS := 1);
IF Axis1_SVON.DONE THEN Axes_SVON_Cmd := FALSE; END_IF;

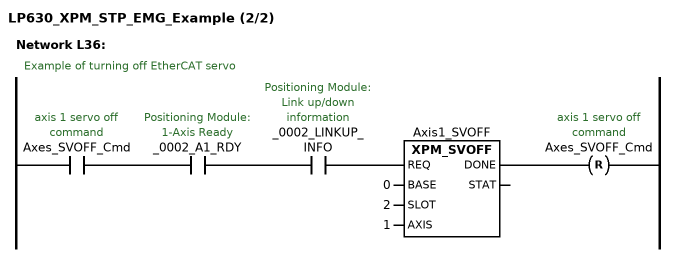
(* Example of turning off EtherCAT servo *)
(* Rung L36 *)
Axis1_SVOFF(REQ := Axes_SVOFF_Cmd AND _0002_A1_RDY AND _0002_LINKUP_INFO, BASE := 0, SLOT := 2, AXIS := 1);
IF Axis1_SVOFF.DONE THEN Axes_SVOFF_Cmd := FALSE; END_IF;
END_PROGRAM

PROGRAM LP631_LinearInterpolation_Example (* task: Scan Program *)
(* example program for XPM_IST and linear interpolation  function block. *)
VAR
    Axes_SVOFF_Cmd : BOOL; (* axis 1 servo off command *)
    Axes_SVON_Cmd : BOOL; (* axes servo on command *)
    Axis1_CMD_Step : UINT; (* step to run in XPM_IST *)
    Axis1_Home : XPM_FLT; (* direct home of axis 1 *)
    Axis1_IST_CMD : BOOL; (* command to jog axis 1 forward *)
    Axis1_IST_FB : XPM_IST; (* xpm_ist for axis 1 *)
    Axis1_SVOFF : XPM_SVOFF; (* function block for axis 1 servo off *)
    Axis1_SVON : XPM_SVON; (* SVON fb for axis 1 *)
    Axis2_Home : XPM_FLT; (* direct home of axis 1 *)
    Axis2_SVOFF : XPM_SVOFF; (* function block for axis 1 servo off *)
    Axis2_SVON : XPM_SVON; (* SVON fb for axis 1 *)
    Connect_Servos : BOOL; (* command to connect to ECAT servos *)
    DCON_FB : XPM_DCON; (* EtherCAT disconnect FB *)
    Disconnect_Servos : BOOL; (* Disconnect from ECAT servos *)
    ECON_FB : XPM_ECON; (* EtherCAT connect FB *)
    Home_Axes : BOOL; (* home the axes *)
END_VAR
VAR_EXTERNAL
    _0002_A1_RDY : BOOL; (* AT %UX0.2.0 *) (* Positioning Module: 1-Axis Ready *)
    _0002_A2_RDY : BOOL; (* AT %UX0.2.1 *) (* Positioning Module: 2-Axis Ready *)
    _0002_LINKUP_INFO : BOOL; (* AT %UX0.2.14 *) (* Positioning Module: Link up/down information *)
END_VAR
VAR
    _p1 : BOOL;
    _p2 : BOOL;
    _p3 : BOOL;
END_VAR

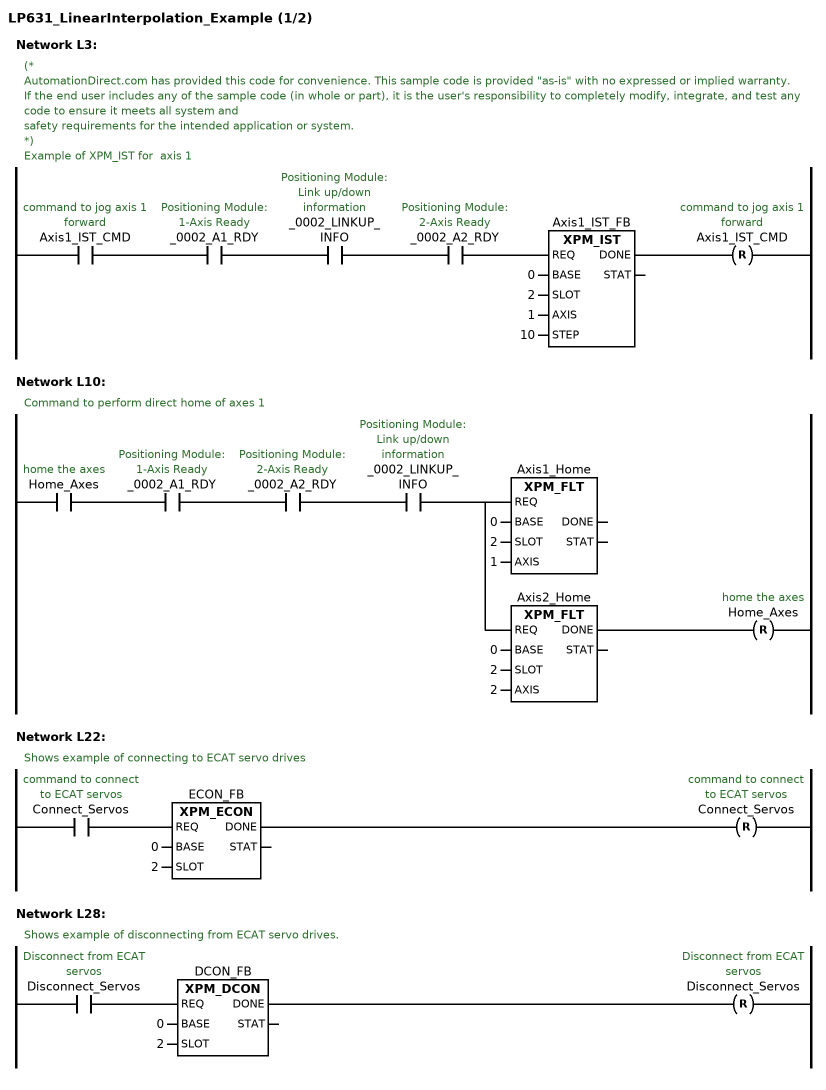
(* ( * / AutomationDirect.com has provided this code for convenience. This sample code is provided "as-is" with no expressed or implied warranty. / If the end user includes any of the sample code (in whole or part), it is the user's responsibility to completely modify, integrate, and test any code to ensure it meets all system and / safety requirements for the intended application or system. / * ) *)
(* Example of XPM_IST for  axis 1 *)
(* Rung L3 *)
Axis1_IST_FB(REQ := Axis1_IST_CMD AND _0002_A1_RDY AND _0002_LINKUP_INFO AND _0002_A2_RDY, BASE := 0, SLOT := 2, AXIS := 1, STEP := 10);
IF Axis1_IST_FB.DONE THEN Axis1_IST_CMD := FALSE; END_IF;
(* Command to perform direct home of axes 1 *)
(* Rung L10 *)
_p1 := Home_Axes AND _0002_A1_RDY AND _0002_A2_RDY AND _0002_LINKUP_INFO;
Axis1_Home(REQ := _p1, BASE := 0, SLOT := 2, AXIS := 1);
Axis2_Home(REQ := _p1, BASE := 0, SLOT := 2, AXIS := 2);
IF Axis2_Home.DONE THEN Home_Axes := FALSE; END_IF;
(* Shows example of connecting to ECAT servo drives *)
(* Rung L22 *)
ECON_FB(REQ := Connect_Servos, BASE := 0, SLOT := 2);
IF ECON_FB.DONE THEN Connect_Servos := FALSE; END_IF;
(* Shows example of disconnecting from ECAT servo drives. *)
(* Rung L28 *)
DCON_FB(REQ := Disconnect_Servos, BASE := 0, SLOT := 2);
IF DCON_FB.DONE THEN Disconnect_Servos := FALSE; END_IF;

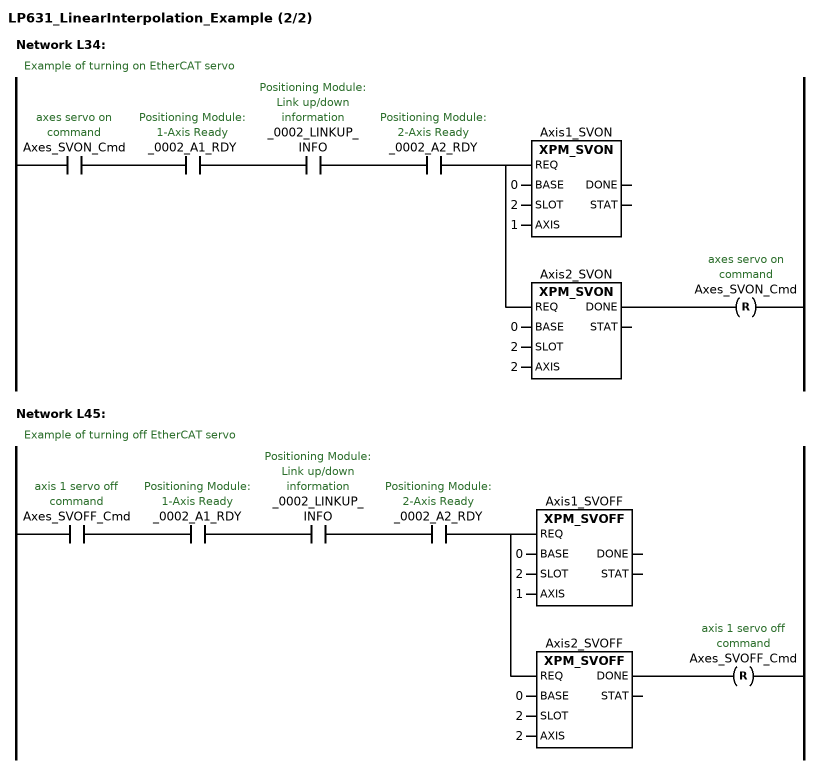
(* Example of turning on EtherCAT servo *)
(* Rung L34 *)
_p2 := Axes_SVON_Cmd AND _0002_A1_RDY AND _0002_LINKUP_INFO AND _0002_A2_RDY;
Axis1_SVON(REQ := _p2, BASE := 0, SLOT := 2, AXIS := 1);
Axis2_SVON(REQ := _p2, BASE := 0, SLOT := 2, AXIS := 2);
IF Axis2_SVON.DONE THEN Axes_SVON_Cmd := FALSE; END_IF;
(* Example of turning off EtherCAT servo *)
(* Rung L45 *)
_p3 := Axes_SVOFF_Cmd AND _0002_A1_RDY AND _0002_LINKUP_INFO AND _0002_A2_RDY;
Axis1_SVOFF(REQ := _p3, BASE := 0, SLOT := 2, AXIS := 1);
Axis2_SVOFF(REQ := _p3, BASE := 0, SLOT := 2, AXIS := 2);
IF Axis2_SVOFF.DONE THEN Axes_SVOFF_Cmd := FALSE; END_IF;
END_PROGRAM

PROGRAM LP632_CircularInterpolation_Example (* task: Scan Program *)
(* example program for XPM_IST and Circular interpolation  function block. *)
VAR
    Axes_SVOFF_Cmd : BOOL; (* axis 1 servo off command *)
    Axes_SVON_Cmd : BOOL; (* axes servo on command *)
    Axis1_CMD_Step : UINT; (* step to run in XPM_IST *)
    Axis1_Home : XPM_FLT; (* direct home of axis 1 *)
    Axis1_IST_CMD : BOOL; (* command to jog axis 1 forward *)
    Axis1_IST_FB : XPM_IST; (* xpm_ist for axis 1 *)
    Axis1_SVOFF : XPM_SVOFF; (* function block for axis 1 servo off *)
    Axis1_SVON : XPM_SVON; (* SVON fb for axis 1 *)
    Axis2_Home : XPM_FLT; (* direct home of axis 1 *)
    Axis2_SVOFF : XPM_SVOFF; (* function block for axis 1 servo off *)
    Axis2_SVON : XPM_SVON; (* SVON fb for axis 1 *)
    Connect_Servos : BOOL; (* command to connect to ECAT servos *)
    DCON_FB : XPM_DCON; (* EtherCAT disconnect FB *)
    Disconnect_Servos : BOOL; (* Disconnect from ECAT servos *)
    ECON_FB : XPM_ECON; (* EtherCAT connect FB *)
    Home_Axes : BOOL; (* home the axes *)
END_VAR
VAR_EXTERNAL
    _0002_A1_RDY : BOOL; (* AT %UX0.2.0 *) (* Positioning Module: 1-Axis Ready *)
    _0002_A2_RDY : BOOL; (* AT %UX0.2.1 *) (* Positioning Module: 2-Axis Ready *)
    _0002_A3_RDY : BOOL; (* AT %UX0.2.2 *) (* Positioning Module: 3-Axis Ready *)
    _0002_LINKUP_INFO : BOOL; (* AT %UX0.2.14 *) (* Positioning Module: Link up/down information *)
END_VAR
VAR
    _p1 : BOOL;
    _p2 : BOOL;
    _p3 : BOOL;
END_VAR

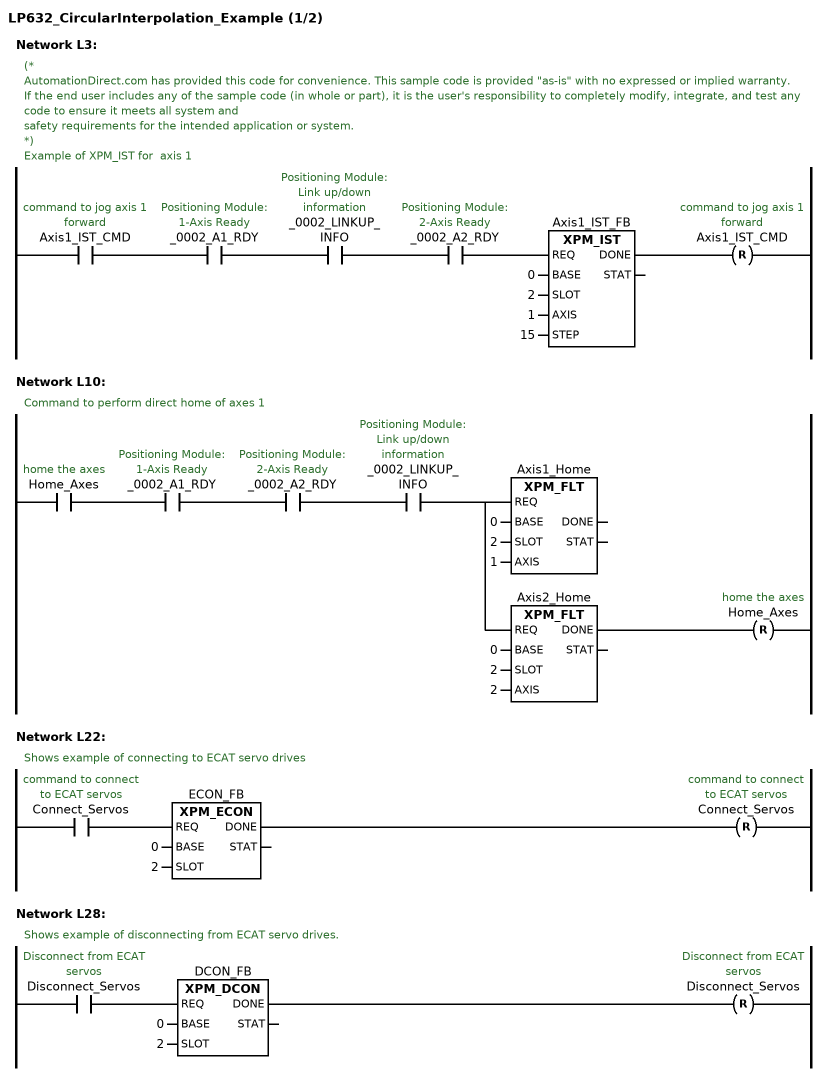
(* ( * / AutomationDirect.com has provided this code for convenience. This sample code is provided "as-is" with no expressed or implied warranty. / If the end user includes any of the sample code (in whole or part), it is the user's responsibility to completely modify, integrate, and test any code to ensure it meets all system and / safety requirements for the intended application or system. / * ) *)
(* Example of XPM_IST for  axis 1 *)
(* Rung L3 *)
Axis1_IST_FB(REQ := Axis1_IST_CMD AND _0002_A1_RDY AND _0002_LINKUP_INFO AND _0002_A2_RDY, BASE := 0, SLOT := 2, AXIS := 1, STEP := 15);
IF Axis1_IST_FB.DONE THEN Axis1_IST_CMD := FALSE; END_IF;
(* Command to perform direct home of axes 1 *)
(* Rung L10 *)
_p1 := Home_Axes AND _0002_A1_RDY AND _0002_A2_RDY AND _0002_LINKUP_INFO;
Axis1_Home(REQ := _p1, BASE := 0, SLOT := 2, AXIS := 1);
Axis2_Home(REQ := _p1, BASE := 0, SLOT := 2, AXIS := 2);
IF Axis2_Home.DONE THEN Home_Axes := FALSE; END_IF;
(* Shows example of connecting to ECAT servo drives *)
(* Rung L22 *)
ECON_FB(REQ := Connect_Servos, BASE := 0, SLOT := 2);
IF ECON_FB.DONE THEN Connect_Servos := FALSE; END_IF;
(* Shows example of disconnecting from ECAT servo drives. *)
(* Rung L28 *)
DCON_FB(REQ := Disconnect_Servos, BASE := 0, SLOT := 2);
IF DCON_FB.DONE THEN Disconnect_Servos := FALSE; END_IF;

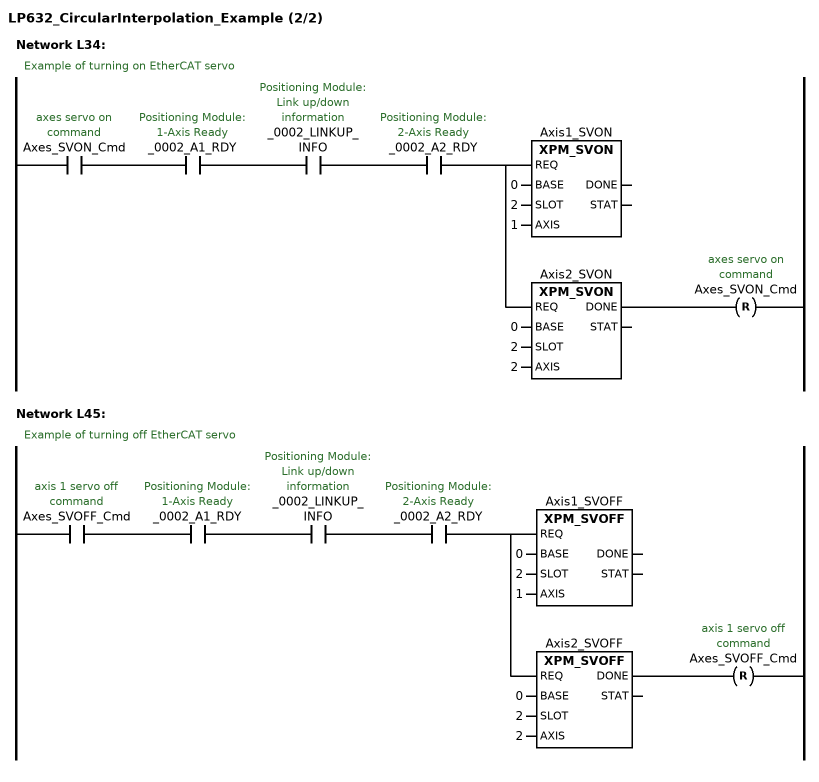
(* Example of turning on EtherCAT servo *)
(* Rung L34 *)
_p2 := Axes_SVON_Cmd AND _0002_A1_RDY AND _0002_LINKUP_INFO AND _0002_A2_RDY;
Axis1_SVON(REQ := _p2, BASE := 0, SLOT := 2, AXIS := 1);
Axis2_SVON(REQ := _p2, BASE := 0, SLOT := 2, AXIS := 2);
IF Axis2_SVON.DONE THEN Axes_SVON_Cmd := FALSE; END_IF;
(* Example of turning off EtherCAT servo *)
(* Rung L45 *)
_p3 := Axes_SVOFF_Cmd AND _0002_A1_RDY AND _0002_LINKUP_INFO AND _0002_A2_RDY;
Axis1_SVOFF(REQ := _p3, BASE := 0, SLOT := 2, AXIS := 1);
Axis2_SVOFF(REQ := _p3, BASE := 0, SLOT := 2, AXIS := 2);
IF Axis2_SVOFF.DONE THEN Axes_SVOFF_Cmd := FALSE; END_IF;
END_PROGRAM

PROGRAM LP633_HelicalInterpolation_Example (* task: Scan Program *)
(* example program for XPM_IST and Helical interpolation  function block. *)
VAR
    Axes_SVOFF_Cmd : BOOL; (* axis 1 servo off command *)
    Axes_SVON_Cmd : BOOL; (* axes servo on command *)
    Axis1_CMD_Step : UINT; (* step to run in XPM_IST *)
    Axis1_Home : XPM_FLT; (* direct home of axis 1 *)
    Axis1_IST_CMD : BOOL; (* command to jog axis 1 forward *)
    Axis1_IST_FB : XPM_IST; (* xpm_ist for axis 1 *)
    Axis1_SVOFF : XPM_SVOFF; (* function block for axis 1 servo off *)
    Axis1_SVON : XPM_SVON; (* SVON fb for axis 1 *)
    Axis2_Home : XPM_FLT; (* direct home of axis 1 *)
    Axis2_SVOFF : XPM_SVOFF; (* function block for axis 1 servo off *)
    Axis2_SVON : XPM_SVON; (* SVON fb for axis 1 *)
    Axis3_Home : XPM_FLT; (* direct home of axis 1 *)
    Axis3_SVOFF : XPM_SVOFF; (* function block for axis 1 servo off *)
    Axis3_SVON : XPM_SVON; (* SVON fb for axis 1 *)
    Connect_Servos : BOOL; (* command to connect to ECAT servos *)
    DCON_FB : XPM_DCON; (* EtherCAT disconnect FB *)
    Disconnect_Servos : BOOL; (* Disconnect from ECAT servos *)
    ECON_FB : XPM_ECON; (* EtherCAT connect FB *)
    Home_Axes : BOOL; (* home the axes *)
END_VAR
VAR_EXTERNAL
    _0002_A1_RDY : BOOL; (* AT %UX0.2.0 *) (* Positioning Module: 1-Axis Ready *)
    _0002_A2_RDY : BOOL; (* AT %UX0.2.1 *) (* Positioning Module: 2-Axis Ready *)
    _0002_A3_RDY : BOOL; (* AT %UX0.2.2 *) (* Positioning Module: 3-Axis Ready *)
    _0002_LINKUP_INFO : BOOL; (* AT %UX0.2.14 *) (* Positioning Module: Link up/down information *)
END_VAR
VAR
    _p1 : BOOL;
    _p2 : BOOL;
    _p3 : BOOL;
END_VAR

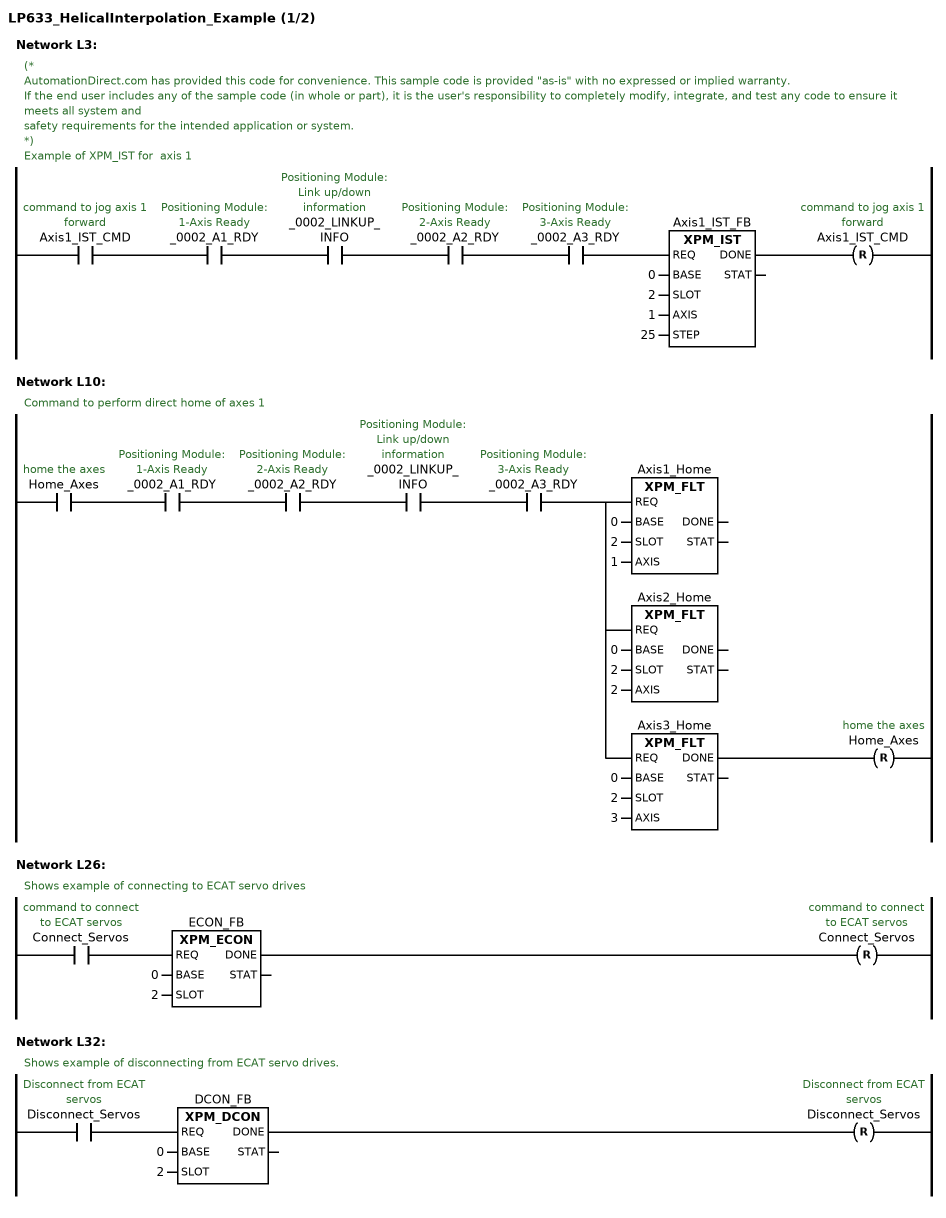
(* ( * / AutomationDirect.com has provided this code for convenience. This sample code is provided "as-is" with no expressed or implied warranty. / If the end user includes any of the sample code (in whole or part), it is the user's responsibility to completely modify, integrate, and test any code to ensure it meets all system and / safety requirements for the intended application or system. / * ) *)
(* Example of XPM_IST for  axis 1 *)
(* Rung L3 *)
Axis1_IST_FB(REQ := Axis1_IST_CMD AND _0002_A1_RDY AND _0002_LINKUP_INFO AND _0002_A2_RDY AND _0002_A3_RDY, BASE := 0, SLOT := 2, AXIS := 1, STEP := 25);
IF Axis1_IST_FB.DONE THEN Axis1_IST_CMD := FALSE; END_IF;
(* Command to perform direct home of axes 1 *)
(* Rung L10 *)
_p1 := Home_Axes AND _0002_A1_RDY AND _0002_A2_RDY AND _0002_LINKUP_INFO AND _0002_A3_RDY;
Axis1_Home(REQ := _p1, BASE := 0, SLOT := 2, AXIS := 1);
Axis2_Home(REQ := _p1, BASE := 0, SLOT := 2, AXIS := 2);
Axis3_Home(REQ := _p1, BASE := 0, SLOT := 2, AXIS := 3);
IF Axis3_Home.DONE THEN Home_Axes := FALSE; END_IF;
(* Shows example of connecting to ECAT servo drives *)
(* Rung L26 *)
ECON_FB(REQ := Connect_Servos, BASE := 0, SLOT := 2);
IF ECON_FB.DONE THEN Connect_Servos := FALSE; END_IF;
(* Shows example of disconnecting from ECAT servo drives. *)
(* Rung L32 *)
DCON_FB(REQ := Disconnect_Servos, BASE := 0, SLOT := 2);
IF DCON_FB.DONE THEN Disconnect_Servos := FALSE; END_IF;

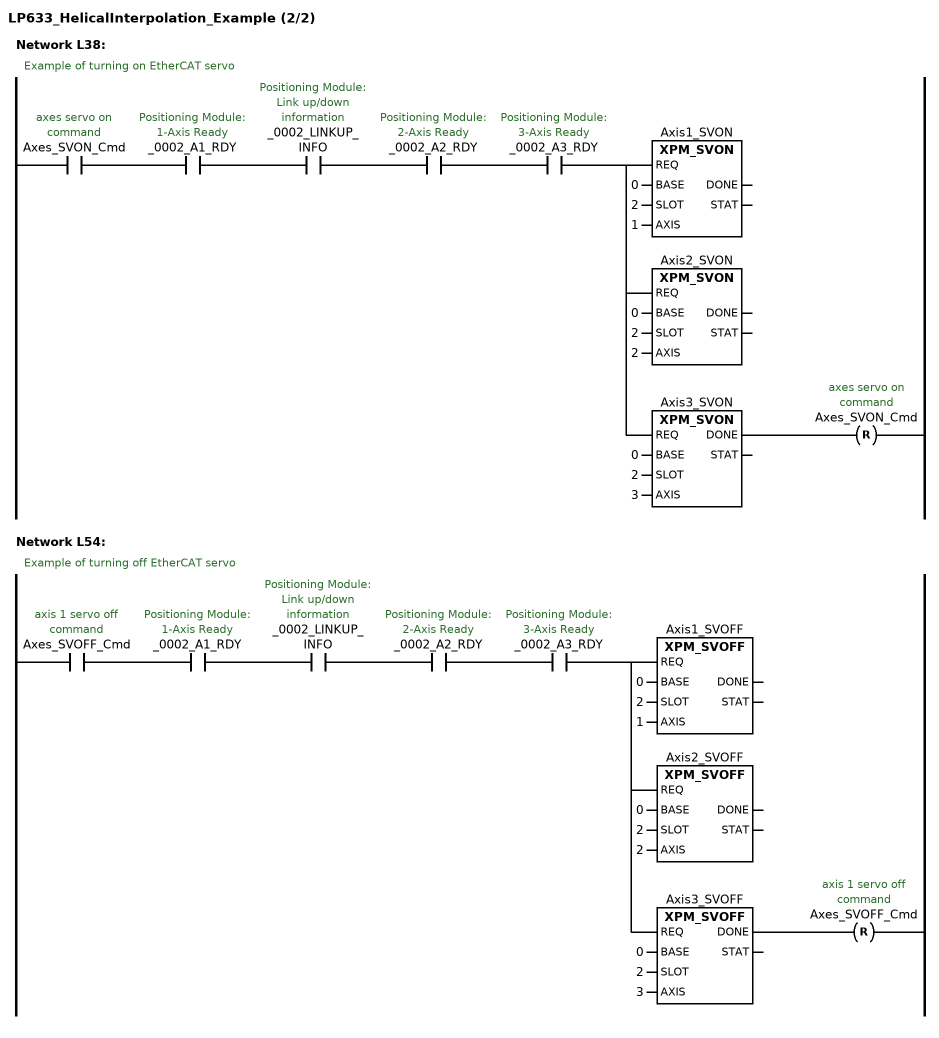
(* Example of turning on EtherCAT servo *)
(* Rung L38 *)
_p2 := Axes_SVON_Cmd AND _0002_A1_RDY AND _0002_LINKUP_INFO AND _0002_A2_RDY AND _0002_A3_RDY;
Axis1_SVON(REQ := _p2, BASE := 0, SLOT := 2, AXIS := 1);
Axis2_SVON(REQ := _p2, BASE := 0, SLOT := 2, AXIS := 2);
Axis3_SVON(REQ := _p2, BASE := 0, SLOT := 2, AXIS := 3);
IF Axis3_SVON.DONE THEN Axes_SVON_Cmd := FALSE; END_IF;
(* Example of turning off EtherCAT servo *)
(* Rung L54 *)
_p3 := Axes_SVOFF_Cmd AND _0002_A1_RDY AND _0002_LINKUP_INFO AND _0002_A2_RDY AND _0002_A3_RDY;
Axis1_SVOFF(REQ := _p3, BASE := 0, SLOT := 2, AXIS := 1);
Axis2_SVOFF(REQ := _p3, BASE := 0, SLOT := 2, AXIS := 2);
Axis3_SVOFF(REQ := _p3, BASE := 0, SLOT := 2, AXIS := 3);
IF Axis3_SVOFF.DONE THEN Axes_SVOFF_Cmd := FALSE; END_IF;
END_PROGRAM

PROGRAM LP634_XPM_SSP_Example (* task: Scan Program *)
(* example program for XPM_SSP *)
VAR
    Axes_SVOFF_Cmd : BOOL; (* axis 1 servo off command *)
    Axes_SVON_Cmd : BOOL; (* axes servo on command *)
    Axis1_Home : XPM_FLT; (* direct home of axis 1 *)
    Axis1_Move_FB : XPM_DST; (* axis 1 speed move fb *)
    Axis1_SVOFF : XPM_SVOFF; (* function block for axis 1 servo off *)
    Axis1_SVON : XPM_SVON; (* SVON fb for axis 1 *)
    Axis2_Home : XPM_FLT; (* direct home of axis 1 *)
    Axis2_SSP_FB : XPM_SSP; (* axis 2 XPM_SSP *)
    Axis2_SVOFF : XPM_SVOFF; (* function block for axis 1 servo off *)
    Axis2_SVON : XPM_SVON; (* SVON fb for axis 1 *)
    Connect_Servos : BOOL; (* command to connect to ECAT servos *)
    DCON_FB : XPM_DCON; (* EtherCAT disconnect FB *)
    Disconnect_Servos : BOOL; (* Disconnect from ECAT servos *)
    ECON_FB : XPM_ECON; (* EtherCAT connect FB *)
    Home_Axes : BOOL; (* home the axes *)
    Run_Example : BOOL; (* command to jog axis 1 forward *)
END_VAR
VAR_EXTERNAL
    _0002_A1_RDY : BOOL; (* AT %UX0.2.0 *) (* Positioning Module: 1-Axis Ready *)
    _0002_A2_RDY : BOOL; (* AT %UX0.2.1 *) (* Positioning Module: 2-Axis Ready *)
    _0002_LINKUP_INFO : BOOL; (* AT %UX0.2.14 *) (* Positioning Module: Link up/down information *)
END_VAR
VAR
    _p1 : BOOL;
    _p2 : BOOL;
    _p3 : BOOL;
    _p4 : BOOL;
END_VAR

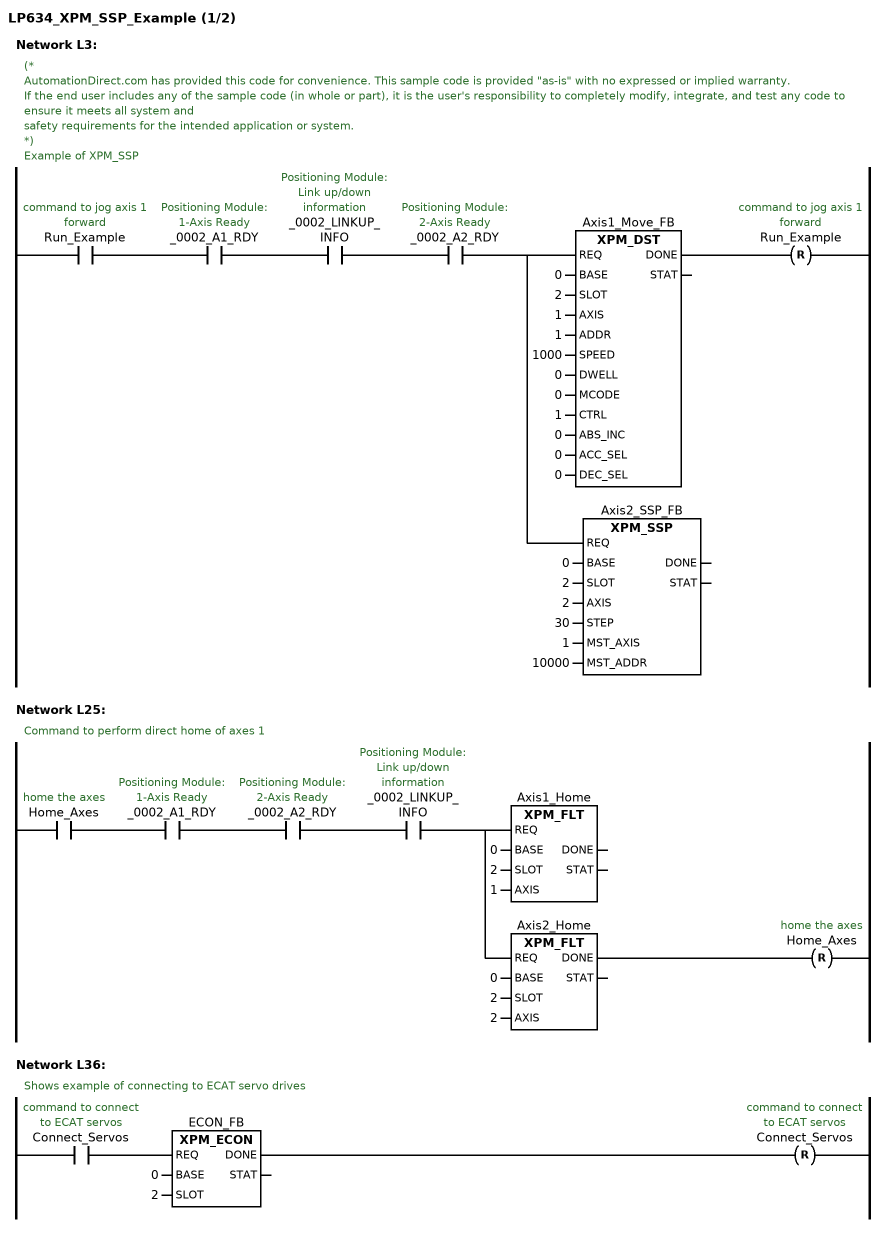
(* ( * / AutomationDirect.com has provided this code for convenience. This sample code is provided "as-is" with no expressed or implied warranty. / If the end user includes any of the sample code (in whole or part), it is the user's responsibility to completely modify, integrate, and test any code to ensure it meets all system and / safety requirements for the intended application or system. / * ) *)
(* Example of XPM_SSP *)
(* Rung L3 *)
_p1 := Run_Example AND _0002_A1_RDY AND _0002_LINKUP_INFO AND _0002_A2_RDY;
Axis1_Move_FB(REQ := _p1, BASE := 0, SLOT := 2, AXIS := 1, ADDR := 1, SPEED := 1000, DWELL := 0, MCODE := 0, CTRL := 1, ABS_INC := 0, ACC_SEL := 0, DEC_SEL := 0);
IF Axis1_Move_FB.DONE THEN Run_Example := FALSE; END_IF;
Axis2_SSP_FB(REQ := _p1, BASE := 0, SLOT := 2, AXIS := 2, STEP := 30, MST_AXIS := 1, MST_ADDR := 10000);
(* Command to perform direct home of axes 1 *)
(* Rung L25 *)
_p2 := Home_Axes AND _0002_A1_RDY AND _0002_A2_RDY AND _0002_LINKUP_INFO;
Axis1_Home(REQ := _p2, BASE := 0, SLOT := 2, AXIS := 1);
Axis2_Home(REQ := _p2, BASE := 0, SLOT := 2, AXIS := 2);
IF Axis2_Home.DONE THEN Home_Axes := FALSE; END_IF;
(* Shows example of connecting to ECAT servo drives *)
(* Rung L36 *)
ECON_FB(REQ := Connect_Servos, BASE := 0, SLOT := 2);
IF ECON_FB.DONE THEN Connect_Servos := FALSE; END_IF;

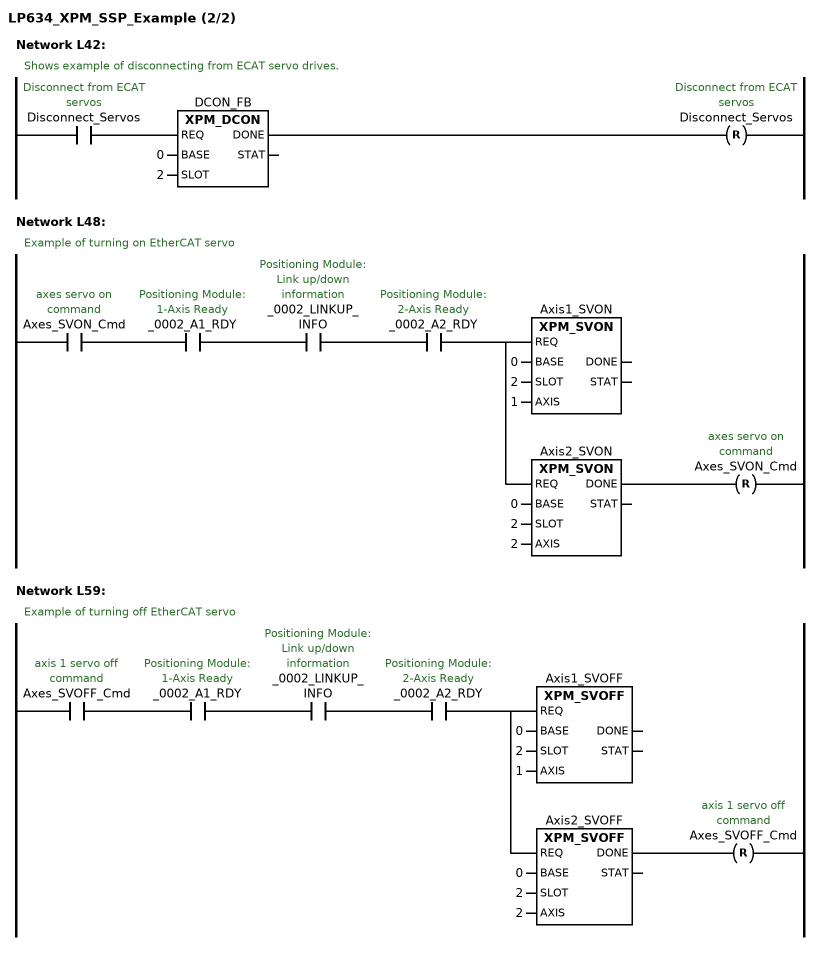
(* Shows example of disconnecting from ECAT servo drives. *)
(* Rung L42 *)
DCON_FB(REQ := Disconnect_Servos, BASE := 0, SLOT := 2);
IF DCON_FB.DONE THEN Disconnect_Servos := FALSE; END_IF;
(* Example of turning on EtherCAT servo *)
(* Rung L48 *)
_p3 := Axes_SVON_Cmd AND _0002_A1_RDY AND _0002_LINKUP_INFO AND _0002_A2_RDY;
Axis1_SVON(REQ := _p3, BASE := 0, SLOT := 2, AXIS := 1);
Axis2_SVON(REQ := _p3, BASE := 0, SLOT := 2, AXIS := 2);
IF Axis2_SVON.DONE THEN Axes_SVON_Cmd := FALSE; END_IF;
(* Example of turning off EtherCAT servo *)
(* Rung L59 *)
_p4 := Axes_SVOFF_Cmd AND _0002_A1_RDY AND _0002_LINKUP_INFO AND _0002_A2_RDY;
Axis1_SVOFF(REQ := _p4, BASE := 0, SLOT := 2, AXIS := 1);
Axis2_SVOFF(REQ := _p4, BASE := 0, SLOT := 2, AXIS := 2);
IF Axis2_SVOFF.DONE THEN Axes_SVOFF_Cmd := FALSE; END_IF;
END_PROGRAM

PROGRAM LP634_XPM_SSS_Example (* task: Scan Program *)
(* example program for XPM_SSS *)
VAR
    Axes_SVOFF_Cmd : BOOL; (* axis 1 servo off command *)
    Axes_SVON_Cmd : BOOL; (* axes servo on command *)
    Axis1_Home : XPM_FLT; (* direct home of axis 1 *)
    Axis1_Move_FB : XPM_DST; (* axis 1 speed move fb *)
    Axis1_SVOFF : XPM_SVOFF; (* function block for axis 1 servo off *)
    Axis1_SVON : XPM_SVON; (* SVON fb for axis 1 *)
    Axis2_Home : XPM_FLT; (* direct home of axis 1 *)
    Axis2_SSS_FB : XPM_SSS; (* axis 2 XPM_SSS fb *)
    Axis2_SVOFF : XPM_SVOFF; (* function block for axis 1 servo off *)
    Axis2_SVON : XPM_SVON; (* SVON fb for axis 1 *)
    Connect_Servos : BOOL; (* command to connect to ECAT servos *)
    DCON_FB : XPM_DCON; (* EtherCAT disconnect FB *)
    Disconnect_Servos : BOOL; (* Disconnect from ECAT servos *)
    ECON_FB : XPM_ECON; (* EtherCAT connect FB *)
    Home_Axes : BOOL; (* home the axes *)
    Run_Example : BOOL; (* command to jog axis 1 forward *)
END_VAR
VAR_EXTERNAL
    _0002_A1_RDY : BOOL; (* AT %UX0.2.0 *) (* Positioning Module: 1-Axis Ready *)
    _0002_A2_RDY : BOOL; (* AT %UX0.2.1 *) (* Positioning Module: 2-Axis Ready *)
    _0002_LINKUP_INFO : BOOL; (* AT %UX0.2.14 *) (* Positioning Module: Link up/down information *)
END_VAR
VAR
    _p1 : BOOL;
    _p2 : BOOL;
    _p3 : BOOL;
    _p4 : BOOL;
END_VAR

